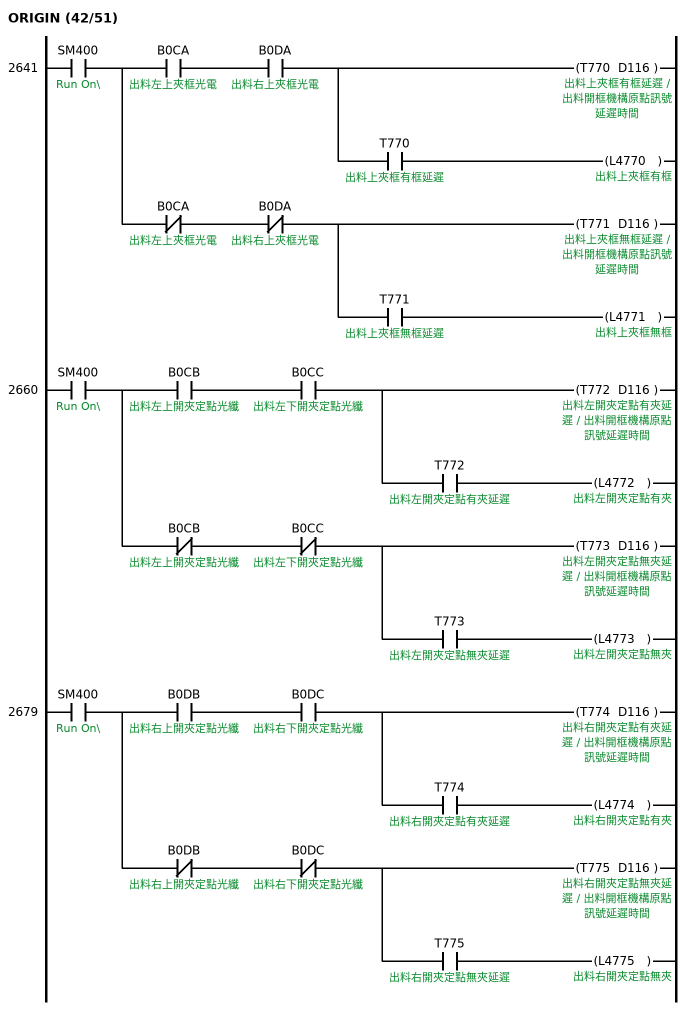
[picture p456: ladder of ORIGIN, rungs at steps 2641 to 2679]
2641  LD      SM400  ; Run On\
      MPS
      AND     B0CA  ; 出料左上夾框光電
      AND     B0DA  ; 出料右上夾框光電
      OUT     T770 D116  ; 出料上夾框有框延遲 / 出料開框機構原點訊號延遲時間
      AND     T770  ; 出料上夾框有框延遲
      OUT     L4770  ; 出料上夾框有框
      MPP
      ANI     B0CA  ; 出料左上夾框光電
      ANI     B0DA  ; 出料右上夾框光電
      OUT     T771 D116  ; 出料上夾框無框延遲 / 出料開框機構原點訊號延遲時間
      AND     T771  ; 出料上夾框無框延遲
      OUT     L4771  ; 出料上夾框無框
2660  LD      SM400  ; Run On\
      MPS
      AND     B0CB  ; 出料左上開夾定點光纖
      AND     B0CC  ; 出料左下開夾定點光纖
      OUT     T772 D116  ; 出料左開夾定點有夾延遲 / 出料開框機構原點訊號延遲時間
      AND     T772  ; 出料左開夾定點有夾延遲
      OUT     L4772  ; 出料左開夾定點有夾
      MPP
      ANI     B0CB  ; 出料左上開夾定點光纖
      ANI     B0CC  ; 出料左下開夾定點光纖
      OUT     T773 D116  ; 出料左開夾定點無夾延遲 / 出料開框機構原點訊號延遲時間
      AND     T773  ; 出料左開夾定點無夾延遲
      OUT     L4773  ; 出料左開夾定點無夾
2679  LD      SM400  ; Run On\
      MPS
      AND     B0DB  ; 出料右上開夾定點光纖
      AND     B0DC  ; 出料右下開夾定點光纖
      OUT     T774 D116  ; 出料右開夾定點有夾延遲 / 出料開框機構原點訊號延遲時間
      AND     T774  ; 出料右開夾定點有夾延遲
      OUT     L4774  ; 出料右開夾定點有夾
      MPP
      ANI     B0DB  ; 出料右上開夾定點光纖
      ANI     B0DC  ; 出料右下開夾定點光纖
      OUT     T775 D116  ; 出料右開夾定點無夾延遲 / 出料開框機構原點訊號延遲時間
      AND     T775  ; 出料右開夾定點無夾延遲
      OUT     L4775  ; 出料右開夾定點無夾
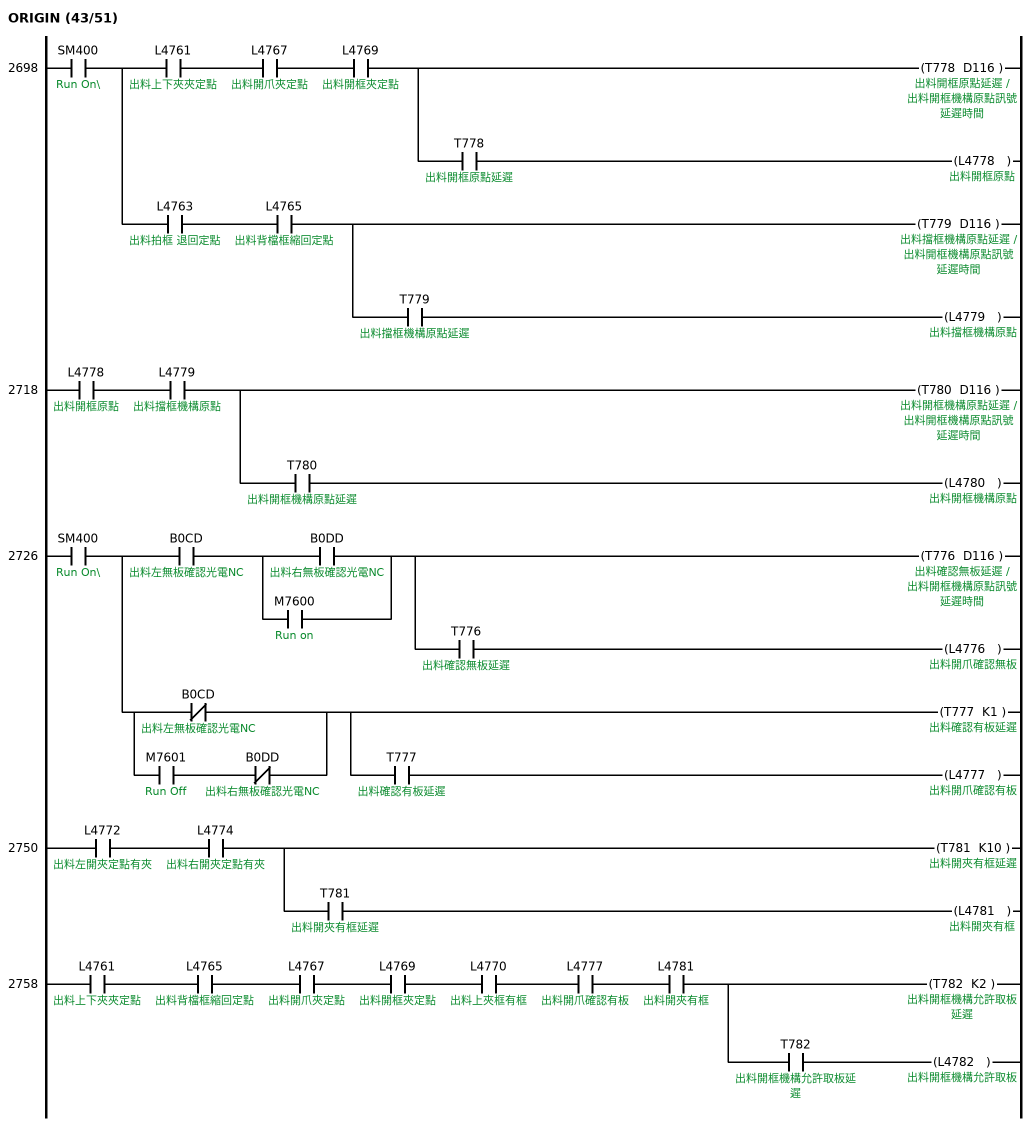
2698  LD      SM400  ; Run On\
      MPS
      AND     L4761  ; 出料上下夾夾定點
      AND     L4767  ; 出料開爪夾定點
      AND     L4769  ; 出料開框夾定點
      OUT     T778 D116  ; 出料開框原點延遲 / 出料開框機構原點訊號延遲時間
      AND     T778  ; 出料開框原點延遲
      OUT     L4778  ; 出料開框原點
      MPP
      AND     L4763  ; 出料拍框 退回定點
      AND     L4765  ; 出料背檔框縮回定點
      OUT     T779 D116  ; 出料擋框機構原點延遲 / 出料開框機構原點訊號延遲時間
      AND     T779  ; 出料擋框機構原點延遲
      OUT     L4779  ; 出料擋框機構原點
2718  LD      L4778  ; 出料開框原點
      AND     L4779  ; 出料擋框機構原點
      OUT     T780 D116  ; 出料開框機構原點延遲 / 出料開框機構原點訊號延遲時間
      AND     T780  ; 出料開框機構原點延遲
      OUT     L4780  ; 出料開框機構原點
2726  LD      SM400  ; Run On\
      MPS
      AND     B0CD  ; 出料左無板確認光電NC
      LD      B0DD  ; 出料右無板確認光電NC
      OR      M7600  ; Run on
      ANB
      OUT     T776 D116  ; 出料確認無板延遲 / 出料開框機構原點訊號延遲時間
      AND     T776  ; 出料確認無板延遲
      OUT     L4776  ; 出料開爪確認無板
      MPP
      LDI     B0CD  ; 出料左無板確認光電NC
      LD      M7601  ; Run Off
      ANI     B0DD  ; 出料右無板確認光電NC
      ORB
      ANB
      OUT     T777 K1  ; 出料確認有板延遲
      AND     T777  ; 出料確認有板延遲
      OUT     L4777  ; 出料開爪確認有板
2750  LD      L4772  ; 出料左開夾定點有夾
      AND     L4774  ; 出料右開夾定點有夾
      OUT     T781 K10  ; 出料開夾有框延遲
      AND     T781  ; 出料開夾有框延遲
      OUT     L4781  ; 出料開夾有框
2758  LD      L4761  ; 出料上下夾夾定點
      AND     L4765  ; 出料背檔框縮回定點
      AND     L4767  ; 出料開爪夾定點
      AND     L4769  ; 出料開框夾定點
      AND     L4770  ; 出料上夾框有框
      AND     L4777  ; 出料開爪確認有板
      AND     L4781  ; 出料開夾有框
      OUT     T782 K2  ; 出料開框機構允許取板延遲
      AND     T782  ; 出料開框機構允許取板延遲
      OUT     L4782  ; 出料開框機構允許取板
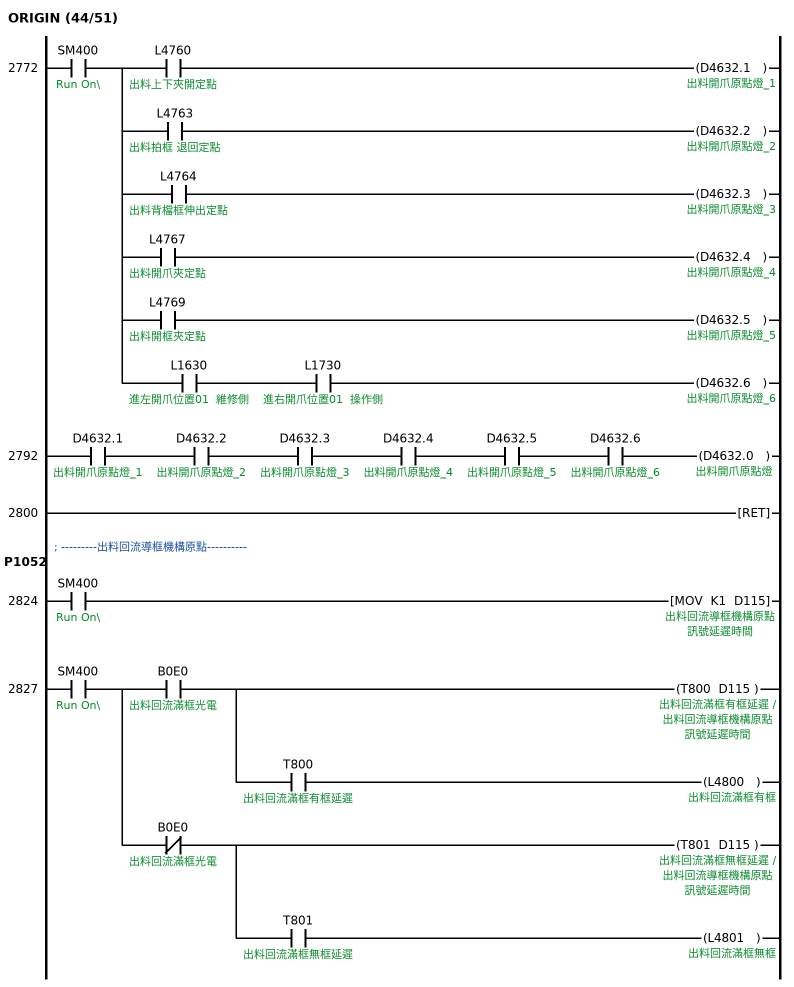
2772  LD      SM400  ; Run On\
      MPS
      AND     L4760  ; 出料上下夾開定點
      OUT     D4632.1  ; 出料開爪原點燈_1
      MRD
      AND     L4763  ; 出料拍框 退回定點
      OUT     D4632.2  ; 出料開爪原點燈_2
      MRD
      AND     L4764  ; 出料背檔框伸出定點
      OUT     D4632.3  ; 出料開爪原點燈_3
      MRD
      AND     L4767  ; 出料開爪夾定點
      OUT     D4632.4  ; 出料開爪原點燈_4
      MRD
      AND     L4769  ; 出料開框夾定點
      OUT     D4632.5  ; 出料開爪原點燈_5
      MPP
      AND     L1630  ; 進左開爪位置01  維修側
      AND     L1730  ; 進右開爪位置01  操作側
      OUT     D4632.6  ; 出料開爪原點燈_6
2792  LD      D4632.1  ; 出料開爪原點燈_1
      AND     D4632.2  ; 出料開爪原點燈_2
      AND     D4632.3  ; 出料開爪原點燈_3
      AND     D4632.4  ; 出料開爪原點燈_4
      AND     D4632.5  ; 出料開爪原點燈_5
      AND     D4632.6  ; 出料開爪原點燈_6
      OUT     D4632.0  ; 出料開爪原點燈
2800  RET
; ---------出料回流導框機構原點----------
      P1052
2824  LD      SM400  ; Run On\
      MOV     K1 D115  ; 出料回流導框機構原點訊號延遲時間
2827  LD      SM400  ; Run On\
      MPS
      AND     B0E0  ; 出料回流滿框光電
      OUT     T800 D115  ; 出料回流滿框有框延遲 / 出料回流導框機構原點訊號延遲時間
      AND     T800  ; 出料回流滿框有框延遲
      OUT     L4800  ; 出料回流滿框有框
      MPP
      ANI     B0E0  ; 出料回流滿框光電
      OUT     T801 D115  ; 出料回流滿框無框延遲 / 出料回流導框機構原點訊號延遲時間
      AND     T801  ; 出料回流滿框無框延遲
      OUT     L4801  ; 出料回流滿框無框
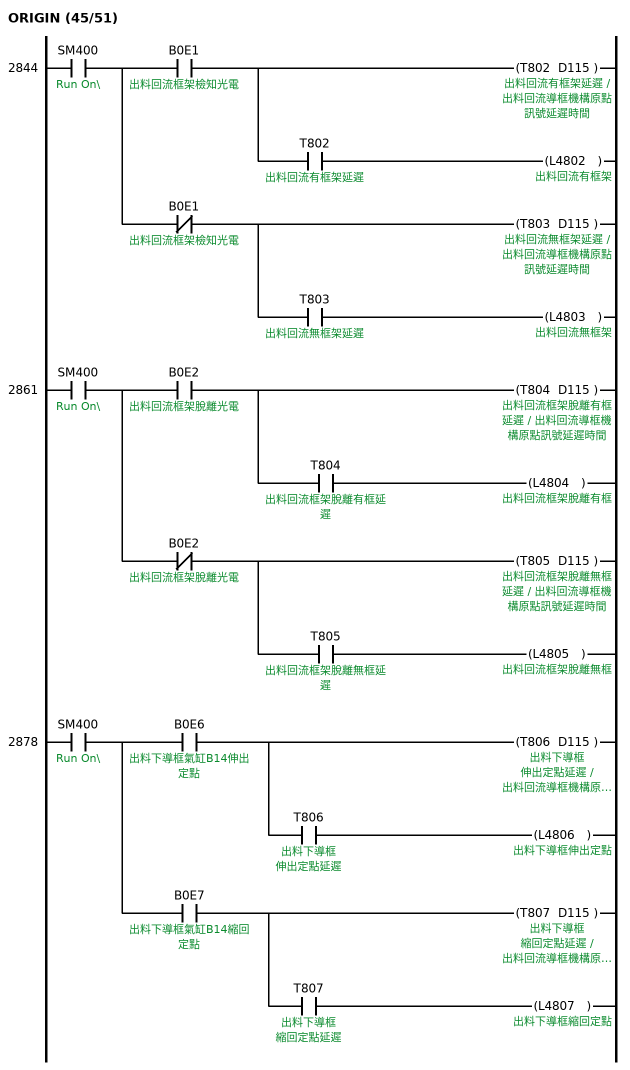
2844  LD      SM400  ; Run On\
      MPS
      AND     B0E1  ; 出料回流框架檢知光電
      OUT     T802 D115  ; 出料回流有框架延遲 / 出料回流導框機構原點訊號延遲時間
      AND     T802  ; 出料回流有框架延遲
      OUT     L4802  ; 出料回流有框架
      MPP
      ANI     B0E1  ; 出料回流框架檢知光電
      OUT     T803 D115  ; 出料回流無框架延遲 / 出料回流導框機構原點訊號延遲時間
      AND     T803  ; 出料回流無框架延遲
      OUT     L4803  ; 出料回流無框架
2861  LD      SM400  ; Run On\
      MPS
      AND     B0E2  ; 出料回流框架脫離光電
      OUT     T804 D115  ; 出料回流框架脫離有框延遲 / 出料回流導框機構原點訊號延遲時間
      AND     T804  ; 出料回流框架脫離有框延遲
      OUT     L4804  ; 出料回流框架脫離有框
      MPP
      ANI     B0E2  ; 出料回流框架脫離光電
      OUT     T805 D115  ; 出料回流框架脫離無框延遲 / 出料回流導框機構原點訊號延遲時間
      AND     T805  ; 出料回流框架脫離無框延遲
      OUT     L4805  ; 出料回流框架脫離無框
2878  LD      SM400  ; Run On\
      MPS
      AND     B0E6  ; 出料下導框氣缸B14伸出定點
      OUT     T806 D115  ; 出料下導框    伸出定點延遲 / 出料回流導框機構原點訊號延遲時間
      AND     T806  ; 出料下導框    伸出定點延遲
      OUT     L4806  ; 出料下導框伸出定點
      MPP
      AND     B0E7  ; 出料下導框氣缸B14縮回定點
      OUT     T807 D115  ; 出料下導框    縮回定點延遲 / 出料回流導框機構原點訊號延遲時間
      AND     T807  ; 出料下導框    縮回定點延遲
      OUT     L4807  ; 出料下導框縮回定點
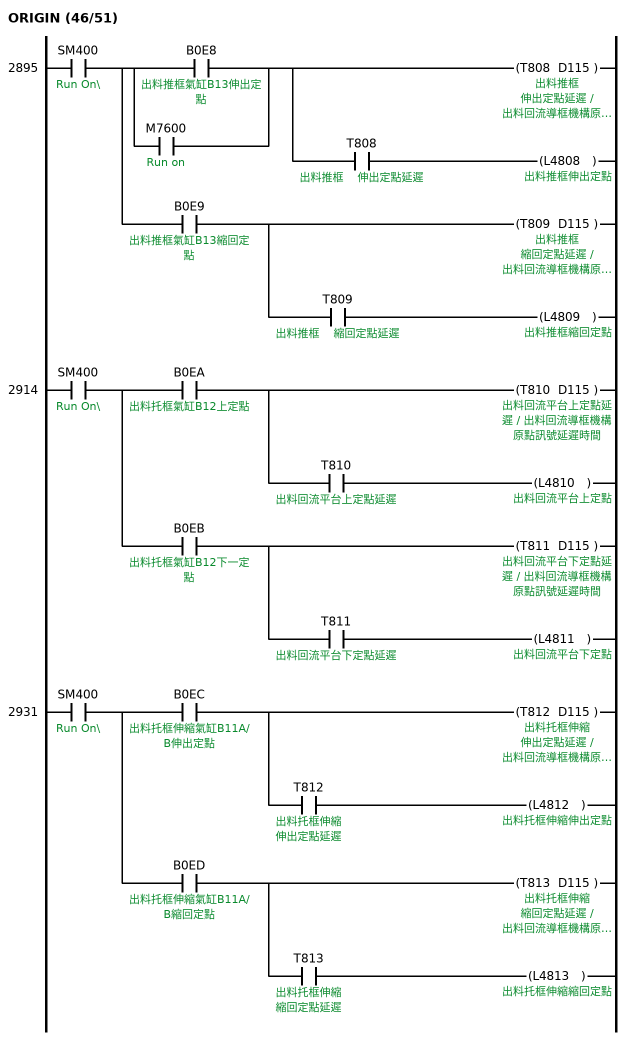
2895  LD      SM400  ; Run On\
      MPS
      LD      B0E8  ; 出料推框氣缸B13伸出定點
      OR      M7600  ; Run on
      ANB
      OUT     T808 D115  ; 出料推框    伸出定點延遲 / 出料回流導框機構原點訊號延遲時間
      AND     T808  ; 出料推框    伸出定點延遲
      OUT     L4808  ; 出料推框伸出定點
      MPP
      AND     B0E9  ; 出料推框氣缸B13縮回定點
      OUT     T809 D115  ; 出料推框    縮回定點延遲 / 出料回流導框機構原點訊號延遲時間
      AND     T809  ; 出料推框    縮回定點延遲
      OUT     L4809  ; 出料推框縮回定點
2914  LD      SM400  ; Run On\
      MPS
      AND     B0EA  ; 出料托框氣缸B12上定點
      OUT     T810 D115  ; 出料回流平台上定點延遲 / 出料回流導框機構原點訊號延遲時間
      AND     T810  ; 出料回流平台上定點延遲
      OUT     L4810  ; 出料回流平台上定點
      MPP
      AND     B0EB  ; 出料托框氣缸B12下一定點
      OUT     T811 D115  ; 出料回流平台下定點延遲 / 出料回流導框機構原點訊號延遲時間
      AND     T811  ; 出料回流平台下定點延遲
      OUT     L4811  ; 出料回流平台下定點
2931  LD      SM400  ; Run On\
      MPS
      AND     B0EC  ; 出料托框伸縮氣缸B11A/B伸出定點
      OUT     T812 D115  ; 出料托框伸縮    伸出定點延遲 / 出料回流導框機構原點訊號延遲時間
      AND     T812  ; 出料托框伸縮    伸出定點延遲
      OUT     L4812  ; 出料托框伸縮伸出定點
      MPP
      AND     B0ED  ; 出料托框伸縮氣缸B11A/B縮回定點
      OUT     T813 D115  ; 出料托框伸縮    縮回定點延遲 / 出料回流導框機構原點訊號延遲時間
      AND     T813  ; 出料托框伸縮    縮回定點延遲
      OUT     L4813  ; 出料托框伸縮縮回定點
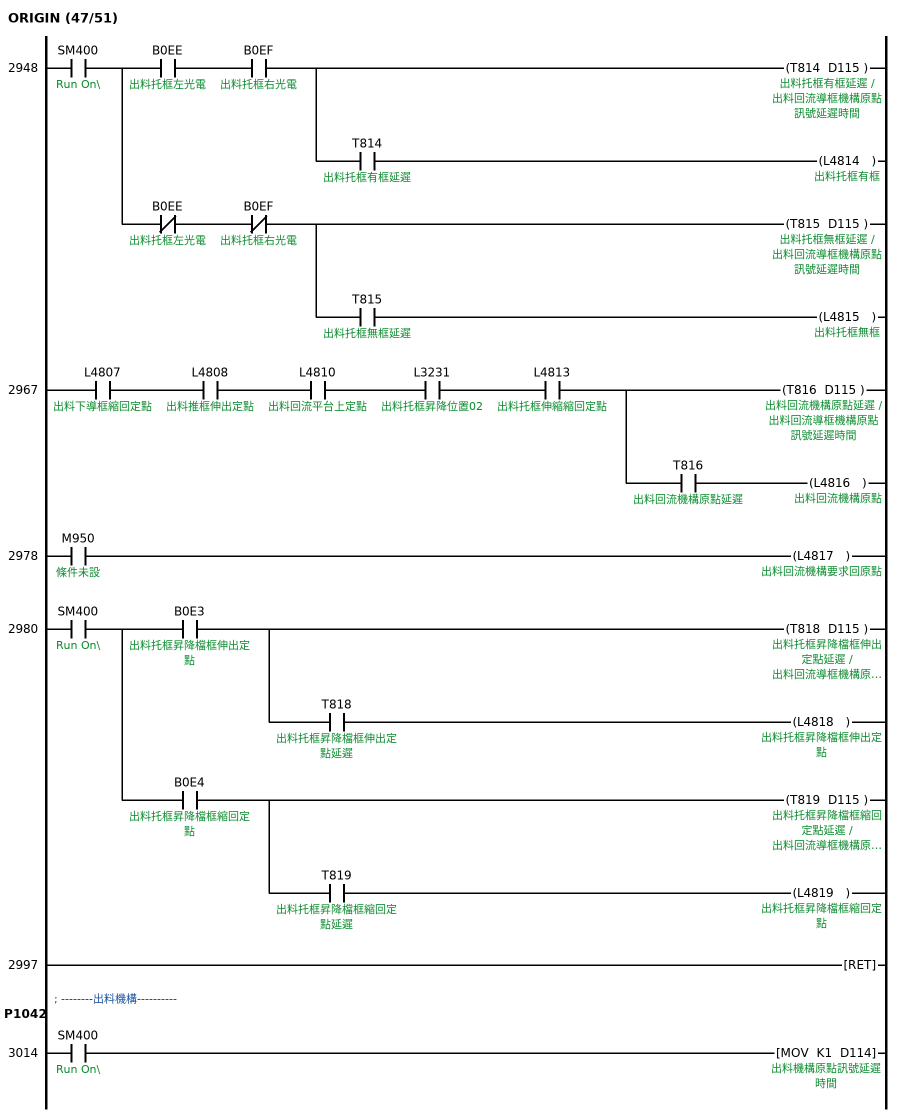
2948  LD      SM400  ; Run On\
      MPS
      AND     B0EE  ; 出料托框左光電
      AND     B0EF  ; 出料托框右光電
      OUT     T814 D115  ; 出料托框有框延遲 / 出料回流導框機構原點訊號延遲時間
      AND     T814  ; 出料托框有框延遲
      OUT     L4814  ; 出料托框有框
      MPP
      ANI     B0EE  ; 出料托框左光電
      ANI     B0EF  ; 出料托框右光電
      OUT     T815 D115  ; 出料托框無框延遲 / 出料回流導框機構原點訊號延遲時間
      AND     T815  ; 出料托框無框延遲
      OUT     L4815  ; 出料托框無框
2967  LD      L4807  ; 出料下導框縮回定點
      AND     L4808  ; 出料推框伸出定點
      AND     L4810  ; 出料回流平台上定點
      AND     L3231  ; 出料托框昇降位置02
      AND     L4813  ; 出料托框伸縮縮回定點
      OUT     T816 D115  ; 出料回流機構原點延遲 / 出料回流導框機構原點訊號延遲時間
      AND     T816  ; 出料回流機構原點延遲
      OUT     L4816  ; 出料回流機構原點
2978  LD      M950  ; 條件未設
      OUT     L4817  ; 出料回流機構要求回原點
2980  LD      SM400  ; Run On\
      MPS
      AND     B0E3  ; 出料托框昇降檔框伸出定點
      OUT     T818 D115  ; 出料托框昇降檔框伸出定點延遲 / 出料回流導框機構原點訊號延遲時間
      AND     T818  ; 出料托框昇降檔框伸出定點延遲
      OUT     L4818  ; 出料托框昇降檔框伸出定點
      MPP
      AND     B0E4  ; 出料托框昇降檔框縮回定點
      OUT     T819 D115  ; 出料托框昇降檔框縮回定點延遲 / 出料回流導框機構原點訊號延遲時間
      AND     T819  ; 出料托框昇降檔框縮回定點延遲
      OUT     L4819  ; 出料托框昇降檔框縮回定點
2997  RET
; --------出料機構----------
      P1042
3014  LD      SM400  ; Run On\
      MOV     K1 D114  ; 出料機構原點訊號延遲時間
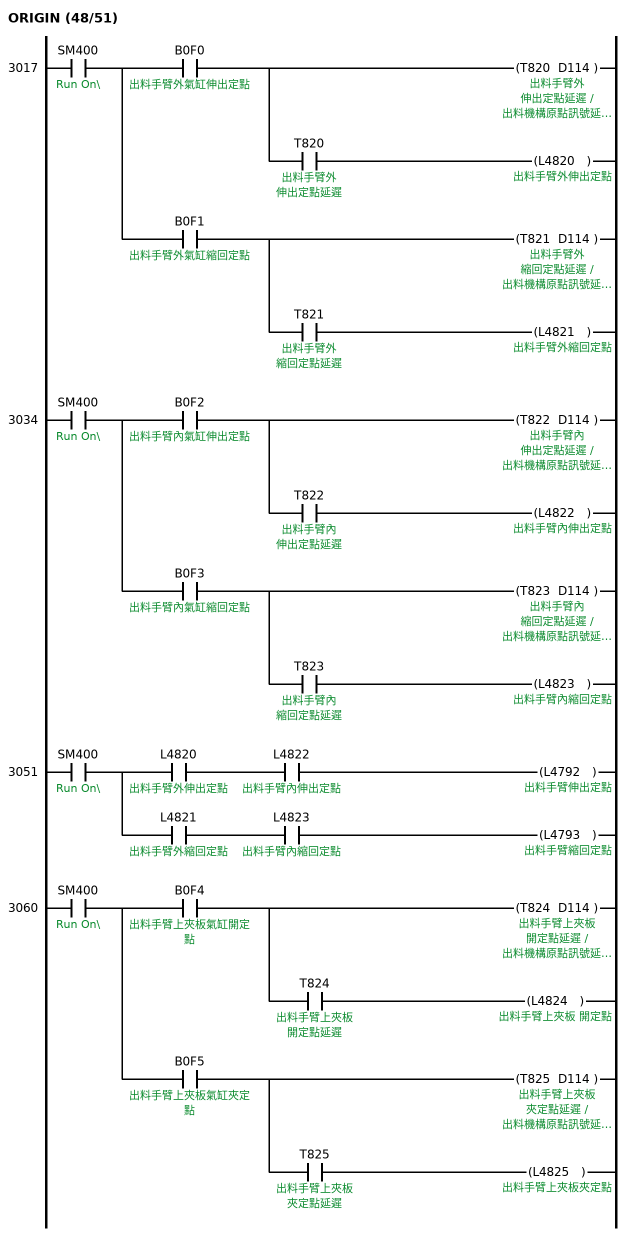
3017  LD      SM400  ; Run On\
      MPS
      AND     B0F0  ; 出料手臂外氣缸伸出定點
      OUT     T820 D114  ; 出料手臂外    伸出定點延遲 / 出料機構原點訊號延遲時間
      AND     T820  ; 出料手臂外    伸出定點延遲
      OUT     L4820  ; 出料手臂外伸出定點
      MPP
      AND     B0F1  ; 出料手臂外氣缸縮回定點
      OUT     T821 D114  ; 出料手臂外    縮回定點延遲 / 出料機構原點訊號延遲時間
      AND     T821  ; 出料手臂外    縮回定點延遲
      OUT     L4821  ; 出料手臂外縮回定點
3034  LD      SM400  ; Run On\
      MPS
      AND     B0F2  ; 出料手臂內氣缸伸出定點
      OUT     T822 D114  ; 出料手臂內    伸出定點延遲 / 出料機構原點訊號延遲時間
      AND     T822  ; 出料手臂內    伸出定點延遲
      OUT     L4822  ; 出料手臂內伸出定點
      MPP
      AND     B0F3  ; 出料手臂內氣缸縮回定點
      OUT     T823 D114  ; 出料手臂內    縮回定點延遲 / 出料機構原點訊號延遲時間
      AND     T823  ; 出料手臂內    縮回定點延遲
      OUT     L4823  ; 出料手臂內縮回定點
3051  LD      SM400  ; Run On\
      MPS
      AND     L4820  ; 出料手臂外伸出定點
      AND     L4822  ; 出料手臂內伸出定點
      OUT     L4792  ; 出料手臂伸出定點
      MPP
      AND     L4821  ; 出料手臂外縮回定點
      AND     L4823  ; 出料手臂內縮回定點
      OUT     L4793  ; 出料手臂縮回定點
3060  LD      SM400  ; Run On\
      MPS
      AND     B0F4  ; 出料手臂上夾板氣缸開定點
      OUT     T824 D114  ; 出料手臂上夾板    開定點延遲 / 出料機構原點訊號延遲時間
      AND     T824  ; 出料手臂上夾板    開定點延遲
      OUT     L4824  ; 出料手臂上夾板 開定點
      MPP
      AND     B0F5  ; 出料手臂上夾板氣缸夾定點
      OUT     T825 D114  ; 出料手臂上夾板    夾定點延遲 / 出料機構原點訊號延遲時間
      AND     T825  ; 出料手臂上夾板    夾定點延遲
      OUT     L4825  ; 出料手臂上夾板夾定點
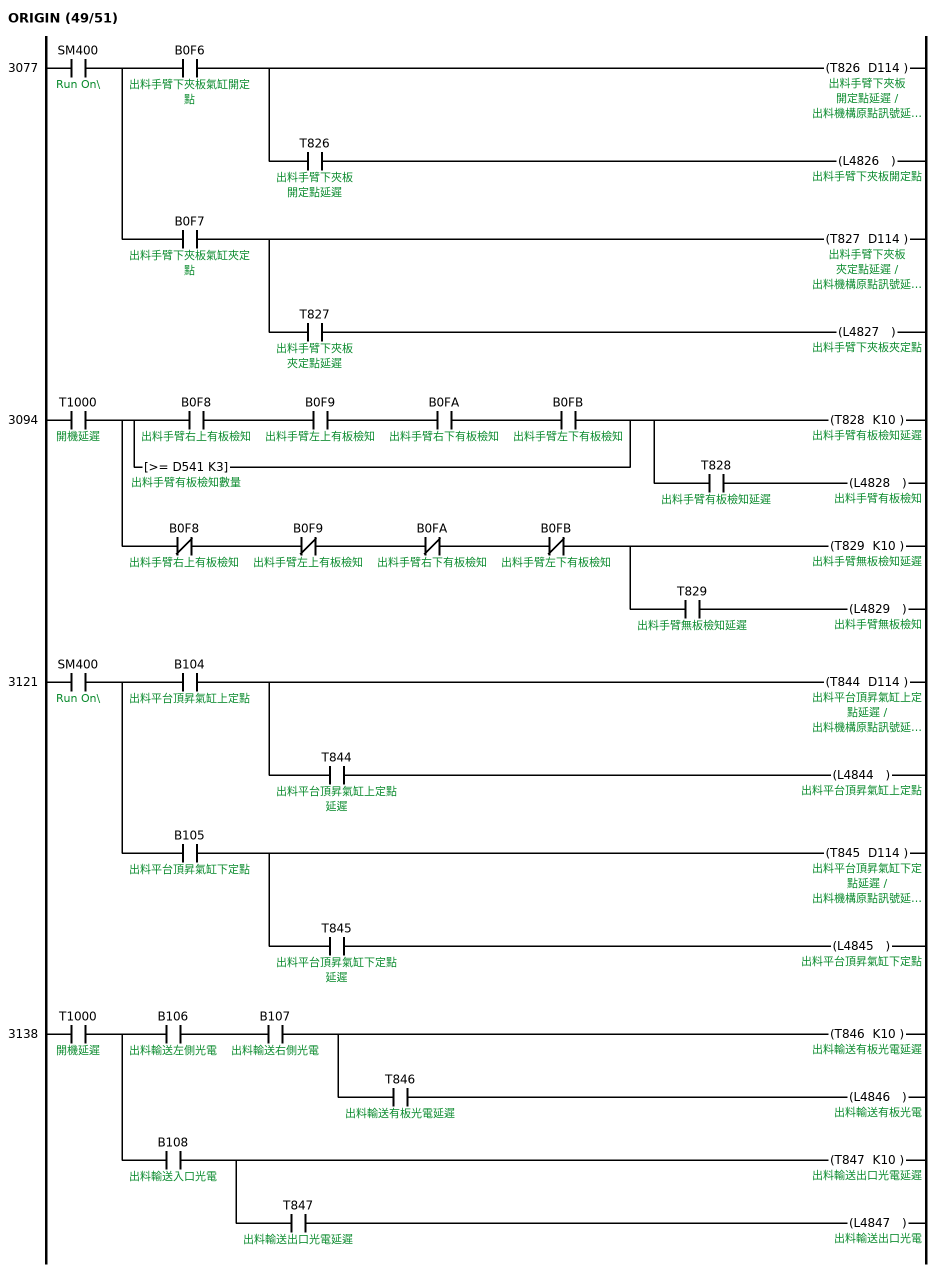
3077  LD      SM400  ; Run On\
      MPS
      AND     B0F6  ; 出料手臂下夾板氣缸開定點
      OUT     T826 D114  ; 出料手臂下夾板    開定點延遲 / 出料機構原點訊號延遲時間
      AND     T826  ; 出料手臂下夾板    開定點延遲
      OUT     L4826  ; 出料手臂下夾板開定點
      MPP
      AND     B0F7  ; 出料手臂下夾板氣缸夾定點
      OUT     T827 D114  ; 出料手臂下夾板    夾定點延遲 / 出料機構原點訊號延遲時間
      AND     T827  ; 出料手臂下夾板    夾定點延遲
      OUT     L4827  ; 出料手臂下夾板夾定點
3094  LD      T1000  ; 開機延遲
      MPS
      LD      B0F8  ; 出料手臂右上有板檢知
      AND     B0F9  ; 出料手臂左上有板檢知
      AND     B0FA  ; 出料手臂右下有板檢知
      AND     B0FB  ; 出料手臂左下有板檢知
      OR>=    D541 K3  ; 出料手臂有板檢知數量
      ANB
      OUT     T828 K10  ; 出料手臂有板檢知延遲
      AND     T828  ; 出料手臂有板檢知延遲
      OUT     L4828  ; 出料手臂有板檢知
      MPP
      ANI     B0F8  ; 出料手臂右上有板檢知
      ANI     B0F9  ; 出料手臂左上有板檢知
      ANI     B0FA  ; 出料手臂右下有板檢知
      ANI     B0FB  ; 出料手臂左下有板檢知
      OUT     T829 K10  ; 出料手臂無板檢知延遲
      AND     T829  ; 出料手臂無板檢知延遲
      OUT     L4829  ; 出料手臂無板檢知
3121  LD      SM400  ; Run On\
      MPS
      AND     B104  ; 出料平台頂昇氣缸上定點
      OUT     T844 D114  ; 出料平台頂昇氣缸上定點延遲 / 出料機構原點訊號延遲時間
      AND     T844  ; 出料平台頂昇氣缸上定點延遲
      OUT     L4844  ; 出料平台頂昇氣缸上定點
      MPP
      AND     B105  ; 出料平台頂昇氣缸下定點
      OUT     T845 D114  ; 出料平台頂昇氣缸下定點延遲 / 出料機構原點訊號延遲時間
      AND     T845  ; 出料平台頂昇氣缸下定點延遲
      OUT     L4845  ; 出料平台頂昇氣缸下定點
3138  LD      T1000  ; 開機延遲
      MPS
      AND     B106  ; 出料輸送左側光電
      AND     B107  ; 出料輸送右側光電
      OUT     T846 K10  ; 出料輸送有板光電延遲
      AND     T846  ; 出料輸送有板光電延遲
      OUT     L4846  ; 出料輸送有板光電
      MPP
      AND     B108  ; 出料輸送入口光電
      OUT     T847 K10  ; 出料輸送出口光電延遲
      AND     T847  ; 出料輸送出口光電延遲
      OUT     L4847  ; 出料輸送出口光電
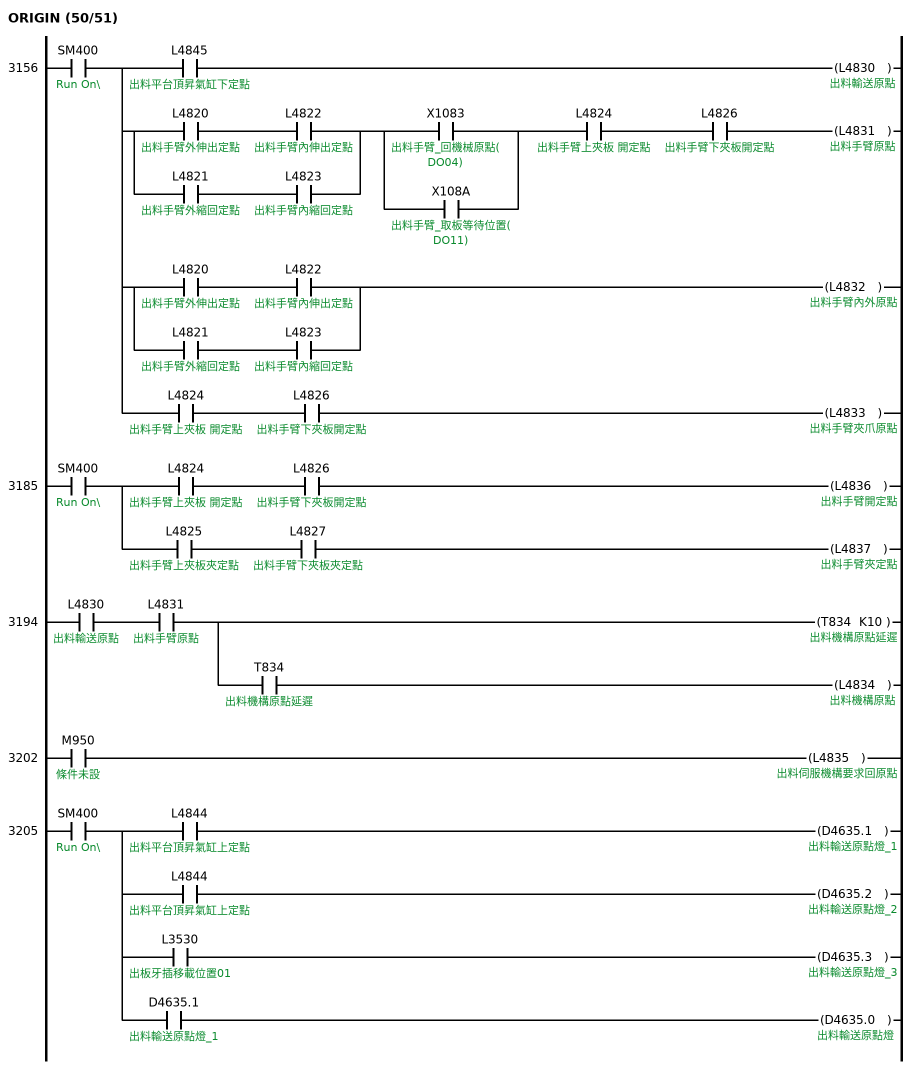
3156  LD      SM400  ; Run On\
      MPS
      AND     L4845  ; 出料平台頂昇氣缸下定點
      OUT     L4830  ; 出料輸送原點
      MRD
      LD      L4820  ; 出料手臂外伸出定點
      AND     L4822  ; 出料手臂內伸出定點
      LD      L4821  ; 出料手臂外縮回定點
      AND     L4823  ; 出料手臂內縮回定點
      ORB
      ANB
      LD      X1083  ; 出料手臂_回機械原點(DO04)
      OR      X108A  ; 出料手臂_取板等待位置(DO11)
      ANB
      AND     L4824  ; 出料手臂上夾板 開定點
      AND     L4826  ; 出料手臂下夾板開定點
      OUT     L4831  ; 出料手臂原點
      MRD
      LD      L4820  ; 出料手臂外伸出定點
      AND     L4822  ; 出料手臂內伸出定點
      LD      L4821  ; 出料手臂外縮回定點
      AND     L4823  ; 出料手臂內縮回定點
      ORB
      ANB
      OUT     L4832  ; 出料手臂內外原點
      MPP
      AND     L4824  ; 出料手臂上夾板 開定點
      AND     L4826  ; 出料手臂下夾板開定點
      OUT     L4833  ; 出料手臂夾爪原點
3185  LD      SM400  ; Run On\
      MPS
      AND     L4824  ; 出料手臂上夾板 開定點
      AND     L4826  ; 出料手臂下夾板開定點
      OUT     L4836  ; 出料手臂開定點
      MPP
      AND     L4825  ; 出料手臂上夾板夾定點
      AND     L4827  ; 出料手臂下夾板夾定點
      OUT     L4837  ; 出料手臂夾定點
3194  LD      L4830  ; 出料輸送原點
      AND     L4831  ; 出料手臂原點
      OUT     T834 K10  ; 出料機構原點延遲
      AND     T834  ; 出料機構原點延遲
      OUT     L4834  ; 出料機構原點
3202  LD      M950  ; 條件未設
      OUT     L4835  ; 出料伺服機構要求回原點
3205  LD      SM400  ; Run On\
      MPS
      AND     L4844  ; 出料平台頂昇氣缸上定點
      OUT     D4635.1  ; 出料輸送原點燈_1
      MRD
      AND     L4844  ; 出料平台頂昇氣缸上定點
      OUT     D4635.2  ; 出料輸送原點燈_2
      MRD
      AND     L3530  ; 出板牙插移載位置01
      OUT     D4635.3  ; 出料輸送原點燈_3
      MPP
      AND     D4635.1  ; 出料輸送原點燈_1
      OUT     D4635.0  ; 出料輸送原點燈
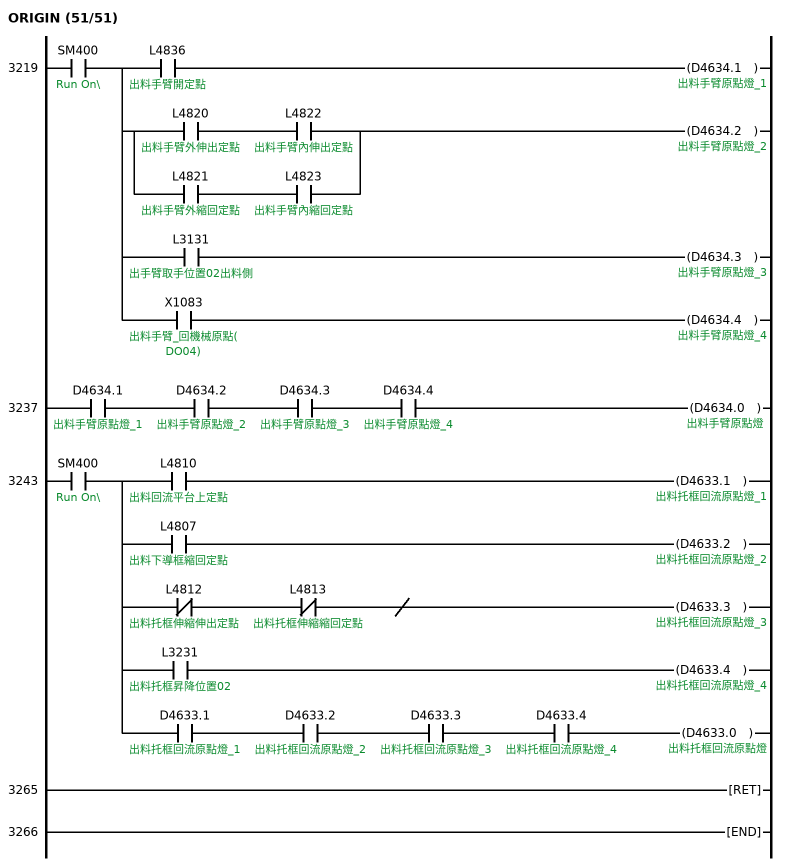
3219  LD      SM400  ; Run On\
      MPS
      AND     L4836  ; 出料手臂開定點
      OUT     D4634.1  ; 出料手臂原點燈_1
      MRD
      LD      L4820  ; 出料手臂外伸出定點
      AND     L4822  ; 出料手臂內伸出定點
      LD      L4821  ; 出料手臂外縮回定點
      AND     L4823  ; 出料手臂內縮回定點
      ORB
      ANB
      OUT     D4634.2  ; 出料手臂原點燈_2
      MRD
      AND     L3131  ; 出手臂取手位置02出料側
      OUT     D4634.3  ; 出料手臂原點燈_3
      MPP
      AND     X1083  ; 出料手臂_回機械原點(DO04)
      OUT     D4634.4  ; 出料手臂原點燈_4
3237  LD      D4634.1  ; 出料手臂原點燈_1
      AND     D4634.2  ; 出料手臂原點燈_2
      AND     D4634.3  ; 出料手臂原點燈_3
      AND     D4634.4  ; 出料手臂原點燈_4
      OUT     D4634.0  ; 出料手臂原點燈
3243  LD      SM400  ; Run On\
      MPS
      AND     L4810  ; 出料回流平台上定點
      OUT     D4633.1  ; 出料托框回流原點燈_1
      MRD
      AND     L4807  ; 出料下導框縮回定點
      OUT     D4633.2  ; 出料托框回流原點燈_2
      MRD
      ANI     L4812  ; 出料托框伸縮伸出定點
      ANI     L4813  ; 出料托框伸縮縮回定點
      INV
      OUT     D4633.3  ; 出料托框回流原點燈_3
      MRD
      AND     L3231  ; 出料托框昇降位置02
      OUT     D4633.4  ; 出料托框回流原點燈_4
      MPP
      AND     D4633.1  ; 出料托框回流原點燈_1
      AND     D4633.2  ; 出料托框回流原點燈_2
      AND     D4633.3  ; 出料托框回流原點燈_3
      AND     D4633.4  ; 出料托框回流原點燈_4
      OUT     D4633.0  ; 出料托框回流原點燈
3265  RET
3266  END
END_PROGRAM

PROGRAM SECS
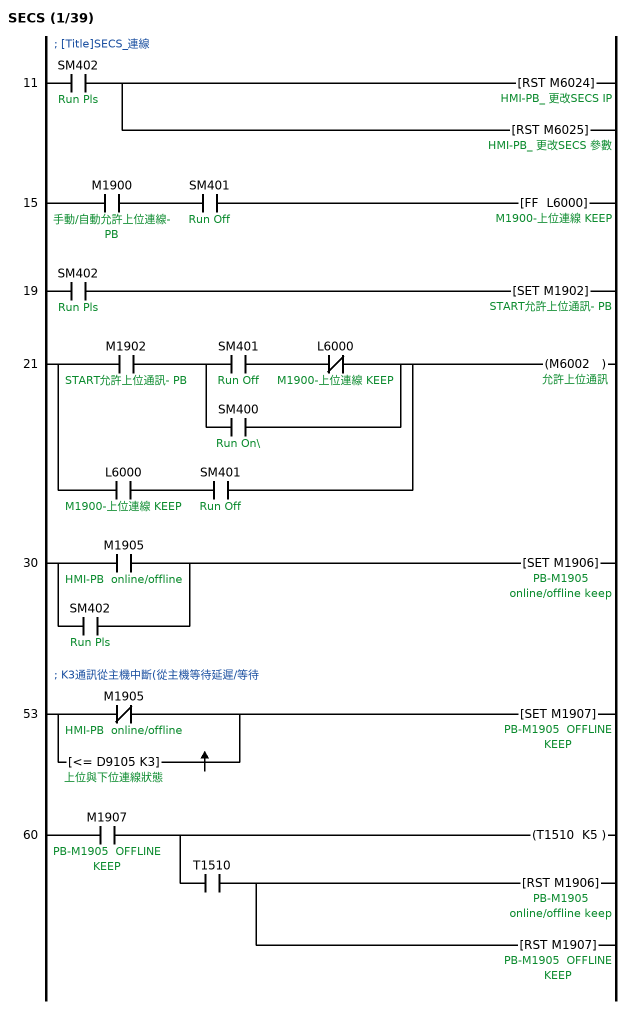
; [Title]SECS_連線
11    LD      SM402  ; Run Pls
      RST     M6024  ; HMI-PB_ 更改SECS IP
      RST     M6025  ; HMI-PB_ 更改SECS 參數
15    LD      M1900  ; 手動/自動允許上位連線-PB
      AND     SM401  ; Run Off
      FF      L6000  ; M1900-上位連線 KEEP
19    LD      SM402  ; Run Pls
      SET     M1902  ; START允許上位通訊- PB
21    LD      M1902  ; START允許上位通訊- PB
      LD      SM401  ; Run Off
      ANI     L6000  ; M1900-上位連線 KEEP
      OR      SM400  ; Run On\
      ANB
      LD      L6000  ; M1900-上位連線 KEEP
      AND     SM401  ; Run Off
      ORB
      OUT     M6002  ; 允許上位通訊
30    LD      M1905  ; HMI-PB  online/offline
      OR      SM402  ; Run Pls
      SET     M1906  ; PB-M1905  online/offline keep
; K3通訊從主機中斷(從主機等待延遲/等待
53    LDI     M1905  ; HMI-PB  online/offline
      LD<=    D9105 K3  ; 上位與下位連線狀態
      MEP
      ORB
      SET     M1907  ; PB-M1905  OFFLINE KEEP
60    LD      M1907  ; PB-M1905  OFFLINE KEEP
      OUT     T1510 K5
      AND     T1510
      RST     M1906  ; PB-M1905  online/offline keep
      RST     M1907  ; PB-M1905  OFFLINE KEEP
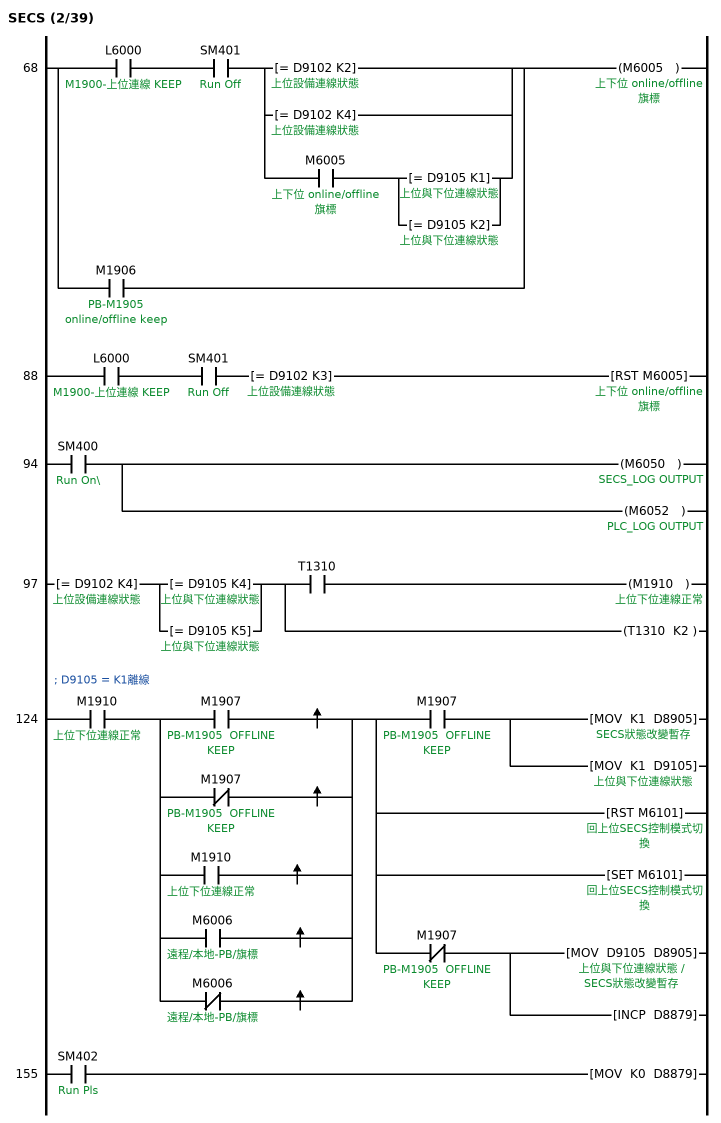
68    LD      L6000  ; M1900-上位連線 KEEP
      AND     SM401  ; Run Off
      LD=     D9102 K2  ; 上位設備連線狀態
      OR=     D9102 K4  ; 上位設備連線狀態
      LD      M6005  ; 上下位 online/offline 旗標
      LD=     D9105 K1  ; 上位與下位連線狀態
      OR=     D9105 K2  ; 上位與下位連線狀態
      ANB
      ORB
      ANB
      OR      M1906  ; PB-M1905  online/offline keep
      OUT     M6005  ; 上下位 online/offline 旗標
88    LD      L6000  ; M1900-上位連線 KEEP
      AND     SM401  ; Run Off
      AND=    D9102 K3  ; 上位設備連線狀態
      RST     M6005  ; 上下位 online/offline 旗標
94    LD      SM400  ; Run On\
      OUT     M6050  ; SECS_LOG OUTPUT
      OUT     M6052  ; PLC_LOG OUTPUT
97    LD=     D9102 K4  ; 上位設備連線狀態
      LD=     D9105 K4  ; 上位與下位連線狀態
      OR=     D9105 K5  ; 上位與下位連線狀態
      ANB
      MPS
      AND     T1310
      OUT     M1910  ; 上位下位連線正常
      MPP
      OUT     T1310 K2
; D9105 = K1離線
124   LD      M1910  ; 上位下位連線正常
      LD      M1907  ; PB-M1905  OFFLINE KEEP
      MEP
      LDI     M1907  ; PB-M1905  OFFLINE KEEP
      MEP
      ORB
      LD      M1910  ; 上位下位連線正常
      MEP
      ORB
      LD      M6006  ; 遠程/本地-PB/旗標
      MEP
      ORB
      LDI     M6006  ; 遠程/本地-PB/旗標
      MEP
      ORB
      ANB
      MPS
      AND     M1907  ; PB-M1905  OFFLINE KEEP
      MOV     K1 D8905  ; SECS狀態改變暫存
      MOV     K1 D9105
      MPP
      RST     M6101  ; 回上位SECS控制模式切換
      SET     M6101  ; 回上位SECS控制模式切換
      ANI     M1907  ; PB-M1905  OFFLINE KEEP
      MOV     D9105 D8905
      INCP    D8879
155   LD      SM402  ; Run Pls
      MOV     K0 D8879
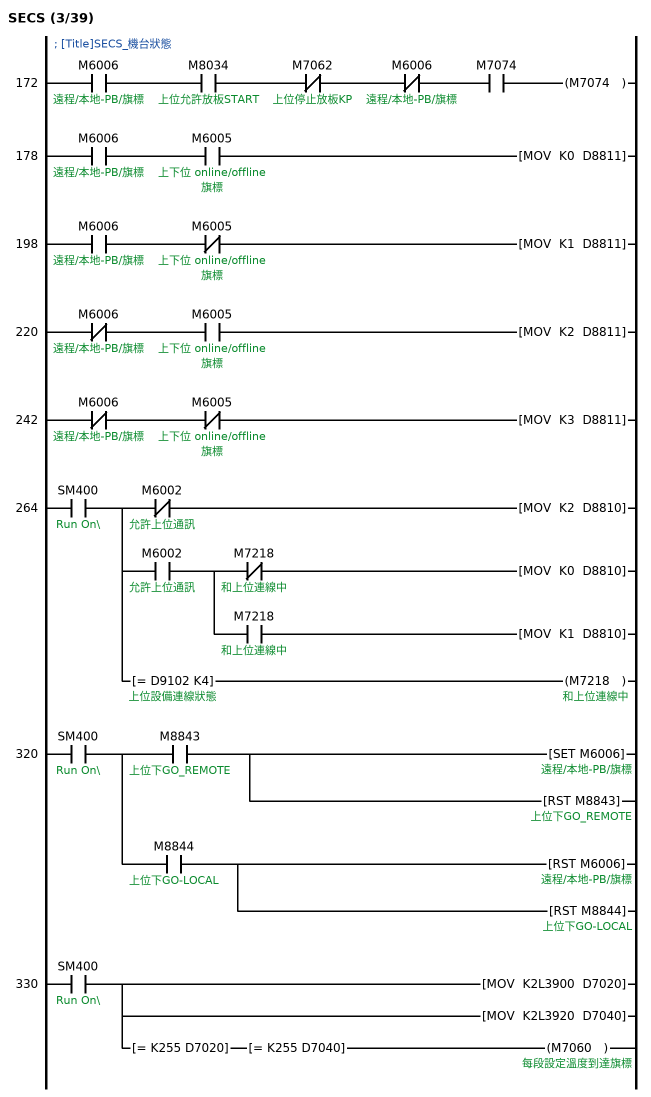
; [Title]SECS_機台狀態
172   LD      M6006  ; 遠程/本地-PB/旗標
      AND     M8034  ; 上位允許放板START
      ANI     M7062  ; 上位停止放板KP
      ANI     M6006  ; 遠程/本地-PB/旗標
      AND     M7074
      OUT     M7074
178   LD      M6006  ; 遠程/本地-PB/旗標
      AND     M6005  ; 上下位 online/offline 旗標
      MOV     K0 D8811
        [note] D8811=K0(遠程控制+SEC在線中)
198   LD      M6006  ; 遠程/本地-PB/旗標
      ANI     M6005  ; 上下位 online/offline 旗標
      MOV     K1 D8811
        [note] D8811= k1(遠程控制中+SEC離線中)
220   LDI     M6006  ; 遠程/本地-PB/旗標
      AND     M6005  ; 上下位 online/offline 旗標
      MOV     K2 D8811
        [note] D881=k2(遠程控制離線+SEC在線中)
242   LDI     M6006  ; 遠程/本地-PB/旗標
      ANI     M6005  ; 上下位 online/offline 旗標
      MOV     K3 D8811
        [note] D881=k3(遠程控制離線+SEC離線中)
264   LD      SM400  ; Run On\
      MPS
      ANI     M6002  ; 允許上位通訊
      MOV     K2 D8810
        [note] K2= SEC通訊未連線
      MRD
      AND     M6002  ; 允許上位通訊
      MPS
      ANI     M7218  ; 和上位連線中
      MOV     K0 D8810
        [note] K0=SEC連線---上位未連線
      MPP
      AND     M7218  ; 和上位連線中
      MOV     K1 D8810
        [note] K1=SEC和上位連線中
      MPP
      AND=    D9102 K4  ; 上位設備連線狀態
      OUT     M7218  ; 和上位連線中
320   LD      SM400  ; Run On\
      MPS
      AND     M8843  ; 上位下GO_REMOTE
      SET     M6006  ; 遠程/本地-PB/旗標
      RST     M8843  ; 上位下GO_REMOTE
      MPP
      AND     M8844  ; 上位下GO-LOCAL
      RST     M6006  ; 遠程/本地-PB/旗標
      RST     M8844  ; 上位下GO-LOCAL
330   LD      SM400  ; Run On\
      MOV     K2L3900 D7020  ; 溫度到達H01
      MOV     K2L3920 D7040  ; 溫度到達IRA01
      AND=    K255 D7020
      AND=    K255 D7040
      OUT     M7060  ; 每段設定溫度到達旗標
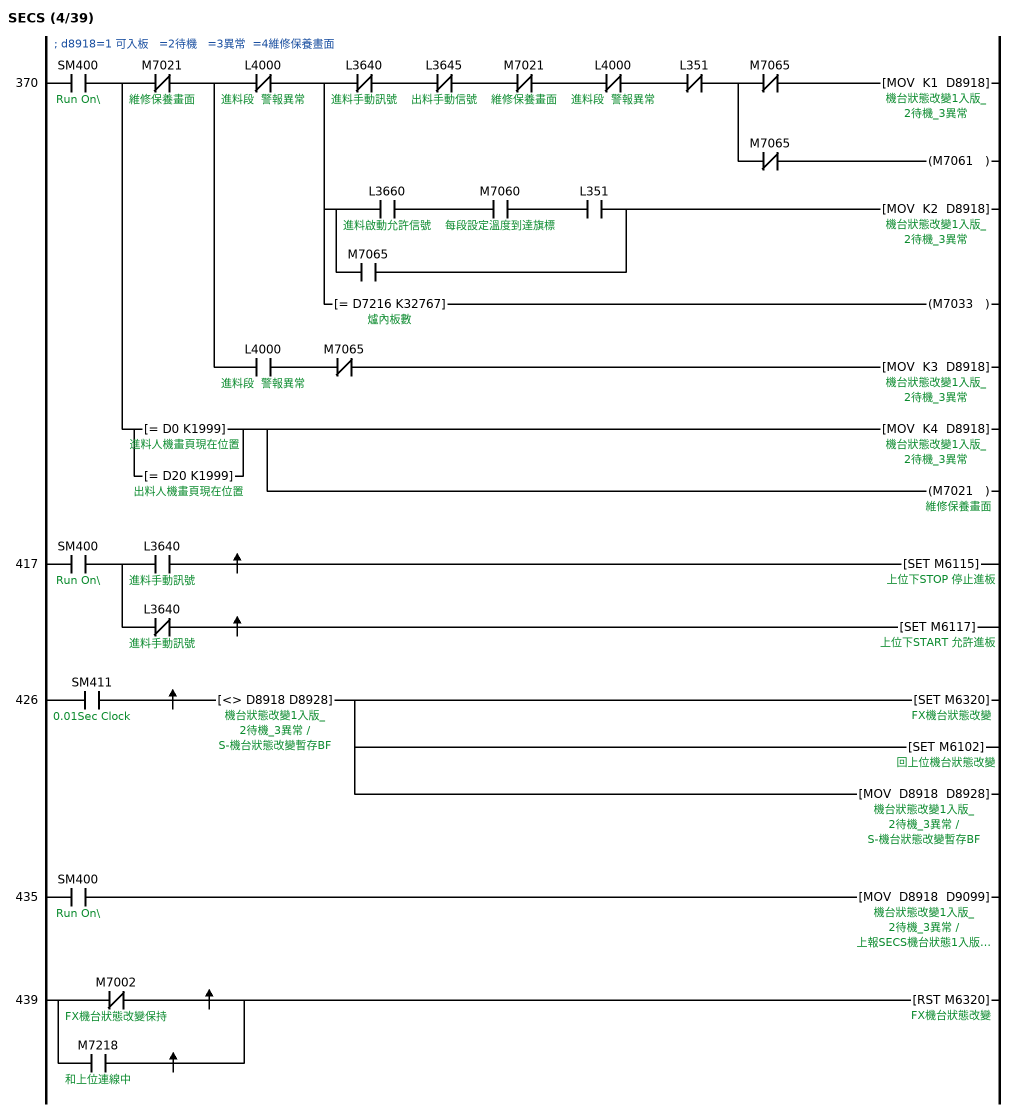
; d8918=1 可入板   =2待機   =3異常  =4維修保養畫面
370   LD      SM400  ; Run On\
      MPS
      ANI     M7021  ; 維修保養畫面
      MPS
      ANI     L4000  ; 進料段  警報異常
      MPS
      ANI     L3640  ; 進料手動訊號
      ANI     L3645  ; 出料手動信號
      ANI     M7021  ; 維修保養畫面
      ANI     L4000  ; 進料段  警報異常
      ANI     L351
      MPS
      ANI     M7065
      MOV     K1 D8918  ; 機台狀態改變1入版_2待機_3異常
      MPP
      ANI     M7065
      OUT     M7061
      MRD
      LD      L3660  ; 進料啟動允許信號
      AND     M7060  ; 每段設定溫度到達旗標
      AND     L351
      OR      M7065
      ANB
      MOV     K2 D8918
      MPP
      AND=    D7216 K32767  ; 爐內板數
      OUT     M7033
      MPP
      AND     L4000  ; 進料段  警報異常
      ANI     M7065
      MOV     K3 D8918
      MPP
      LD=     D0 K1999  ; 進料人機畫頁現在位置
      OR=     D20 K1999  ; 出料人機畫頁現在位置
      ANB
      MOV     K4 D8918
      OUT     M7021  ; 維修保養畫面
417   LD      SM400  ; Run On\
      MPS
      AND     L3640  ; 進料手動訊號
      MEP
      SET     M6115  ; 上位下STOP 停止進板
      MPP
      ANI     L3640  ; 進料手動訊號
      MEP
      SET     M6117  ; 上位下START 允許進板
426   LD      SM411  ; 0.01Sec Clock
      MEP
      AND<>   D8918 D8928  ; 機台狀態改變1入版_2待機_3異常 / S-機台狀態改變暫存BF
      SET     M6320  ; FX機台狀態改變
      SET     M6102  ; 回上位機台狀態改變
      MOV     D8918 D8928
435   LD      SM400  ; Run On\
      MOV     D8918 D9099  ; 上報SECS機台狀態1入版_2待機_3異
439   LDI     M7002  ; FX機台狀態改變保持
      MEP
      LD      M7218  ; 和上位連線中
      MEP
      ORB
      RST     M6320  ; FX機台狀態改變
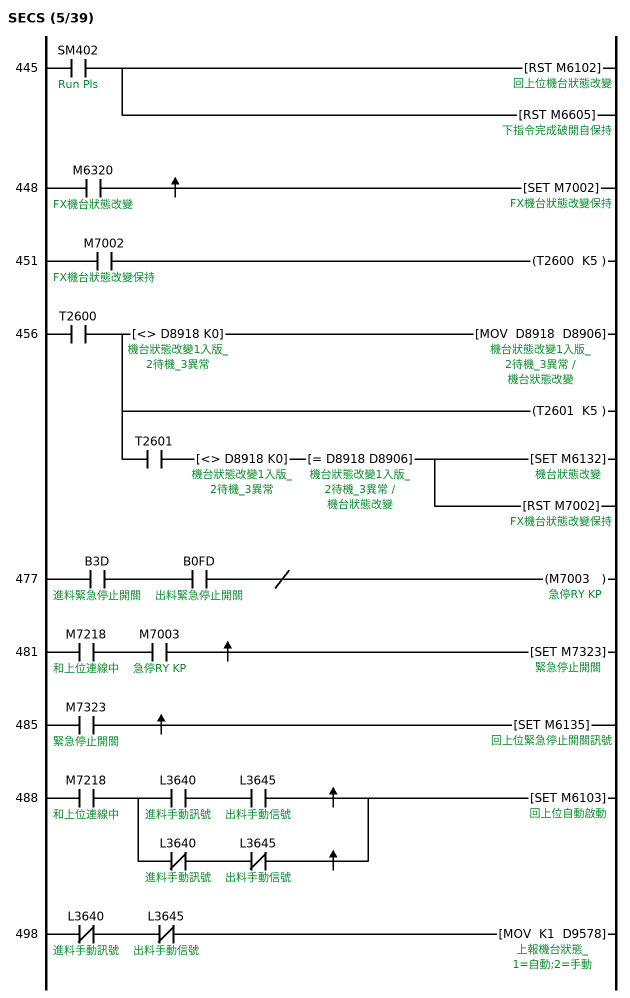
445   LD      SM402  ; Run Pls
      RST     M6102  ; 回上位機台狀態改變
      RST     M6605  ; 下指令完成破開自保持
448   LD      M6320  ; FX機台狀態改變
      MEP
      SET     M7002  ; FX機台狀態改變保持
451   LD      M7002  ; FX機台狀態改變保持
      OUT     T2600 K5
456   LD      T2600
      MPS
      AND<>   D8918 K0  ; 機台狀態改變1入版_2待機_3異常
      MOV     D8918 D8906  ; 機台狀態改變
      MPP
      OUT     T2601 K5
      AND     T2601
      AND<>   D8918 K0  ; 機台狀態改變1入版_2待機_3異常
      AND=    D8918 D8906  ; 機台狀態改變1入版_2待機_3異常 / 機台狀態改變
      SET     M6132  ; 機台狀態改變
      RST     M7002  ; FX機台狀態改變保持
477   LD      B3D  ; 進料緊急停止開關
      AND     B0FD  ; 出料緊急停止開關
      INV
      OUT     M7003  ; 急停RY KP
481   LD      M7218  ; 和上位連線中
      AND     M7003  ; 急停RY KP
      MEP
      SET     M7323  ; 緊急停止開關
485   LD      M7323  ; 緊急停止開關
      MEP
      SET     M6135  ; 回上位緊急停止開關訊號
488   LD      M7218  ; 和上位連線中
      LD      L3640  ; 進料手動訊號
      AND     L3645  ; 出料手動信號
      MEP
      LDI     L3640  ; 進料手動訊號
      ANI     L3645  ; 出料手動信號
      MEP
      ORB
      ANB
      SET     M6103  ; 回上位自動啟動
498   LDI     L3640  ; 進料手動訊號
      ANI     L3645  ; 出料手動信號
      MOV     K1 D9578  ; 上報機台狀態_1=自動;2=手動
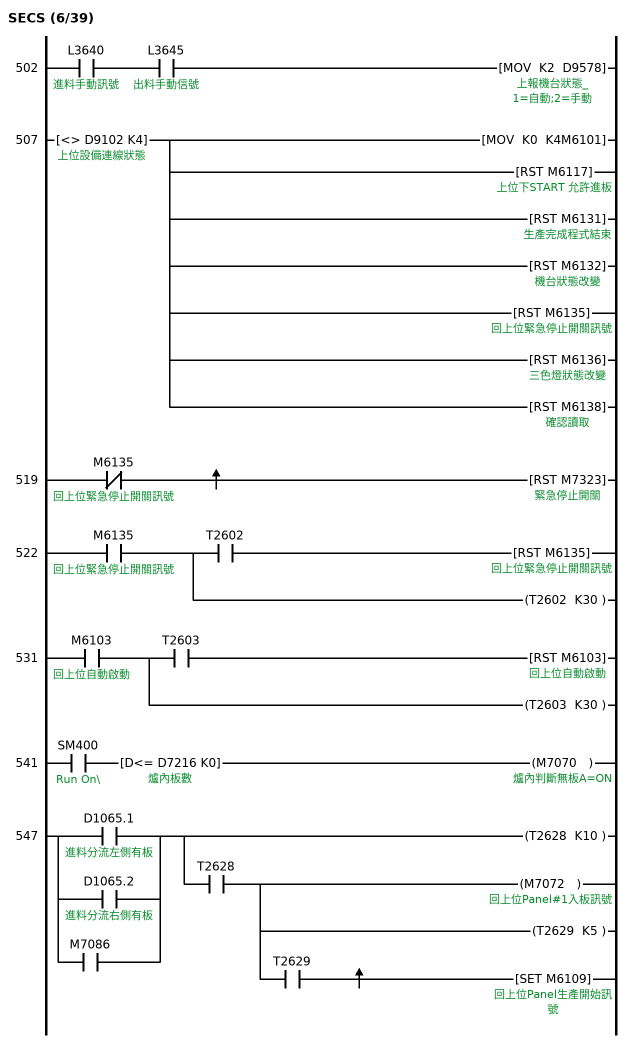
502   LD      L3640  ; 進料手動訊號
      AND     L3645  ; 出料手動信號
      MOV     K2 D9578
507   LD<>    D9102 K4  ; 上位設備連線狀態
      MOV     K0 K4M6101
      RST     M6117  ; 上位下START 允許進板
      RST     M6131  ; 生產完成程式結束
      RST     M6132  ; 機台狀態改變
      RST     M6135  ; 回上位緊急停止開關訊號
      RST     M6136  ; 三色燈狀態改變
      RST     M6138  ; 確認讀取
519   LDI     M6135  ; 回上位緊急停止開關訊號
      MEP
      RST     M7323  ; 緊急停止開關
522   LD      M6135  ; 回上位緊急停止開關訊號
      MPS
      AND     T2602
      RST     M6135  ; 回上位緊急停止開關訊號
      MPP
      OUT     T2602 K30
531   LD      M6103  ; 回上位自動啟動
      MPS
      AND     T2603
      RST     M6103  ; 回上位自動啟動
      MPP
      OUT     T2603 K30
541   LD      SM400  ; Run On\
      ANDD<=  D7216 K0  ; 爐內板數
      OUT     M7070  ; 爐內判斷無板A=ON
547   LD      D1065.1  ; 進料分流左側有板
      OR      D1065.2  ; 進料分流右側有板
      OR      M7086
      OUT     T2628 K10
      AND     T2628
      OUT     M7072  ; 回上位Panel#1入板訊號
      OUT     T2629 K5
      AND     T2629
      MEP
      SET     M6109  ; 回上位Panel生產開始訊號
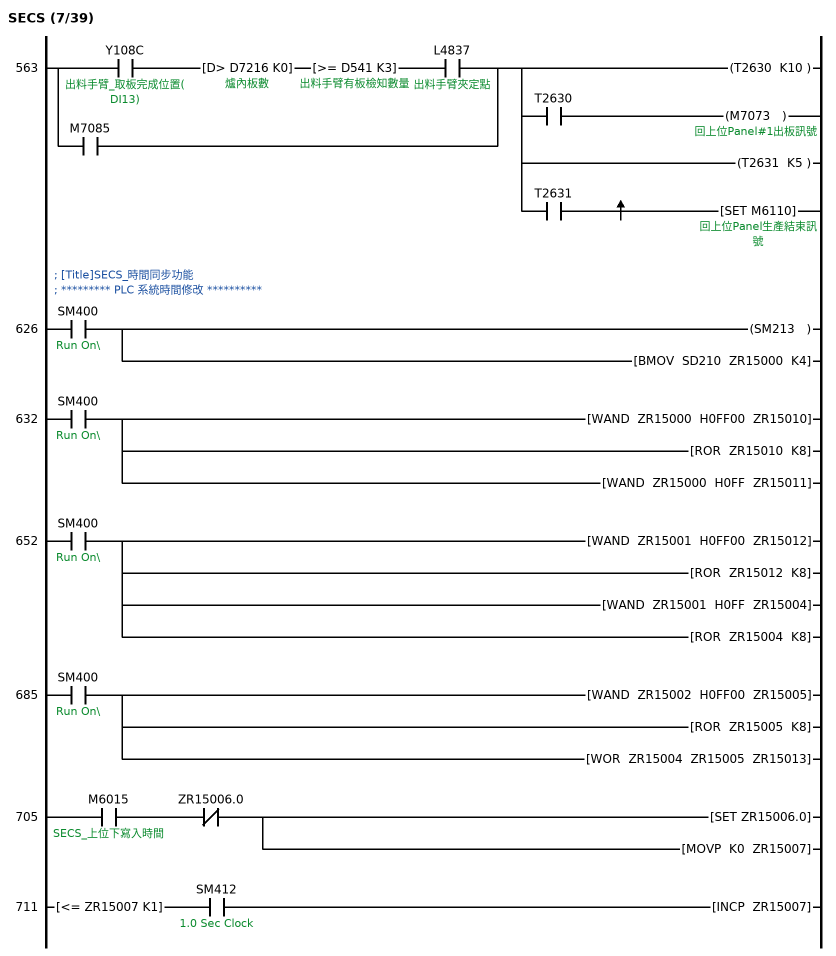
563   LD      Y108C  ; 出料手臂_取板完成位置(DI13)
      ANDD>   D7216 K0  ; 爐內板數
      AND>=   D541 K3  ; 出料手臂有板檢知數量
      AND     L4837  ; 出料手臂夾定點
      OR      M7085
      OUT     T2630 K10
      MPS
      AND     T2630
      OUT     M7073  ; 回上位Panel#1出板訊號
      MPP
      OUT     T2631 K5
      AND     T2631
      MEP
      SET     M6110  ; 回上位Panel生產結束訊號
; [Title]SECS_時間同步功能
; ********* PLC 系統時間修改 **********
626   LD      SM400  ; Run On\
      OUT     SM213
      BMOV    SD210 ZR15000 K4
632   LD      SM400  ; Run On\
      WAND    ZR15000 H0FF00 ZR15010
      ROR     ZR15010 K8
        [note] 高低位資料互換
      WAND    ZR15000 H0FF ZR15011
652   LD      SM400  ; Run On\
      WAND    ZR15001 H0FF00 ZR15012
      ROR     ZR15012 K8
        [note] 高低位資料互換
      WAND    ZR15001 H0FF ZR15004
      ROR     ZR15004 K8
        [note] 高低位資料互換
685   LD      SM400  ; Run On\
      WAND    ZR15002 H0FF00 ZR15005
      ROR     ZR15005 K8
        [note] 高低位資料互換
      WOR     ZR15004 ZR15005 ZR15013
705   LD      M6015  ; SECS_上位下寫入時間
      ANI     ZR15006.0
      SET     ZR15006.0
      MOVP    K0 ZR15007
711   LD<=    ZR15007 K1
      AND     SM412  ; 1.0 Sec Clock
      INCP    ZR15007
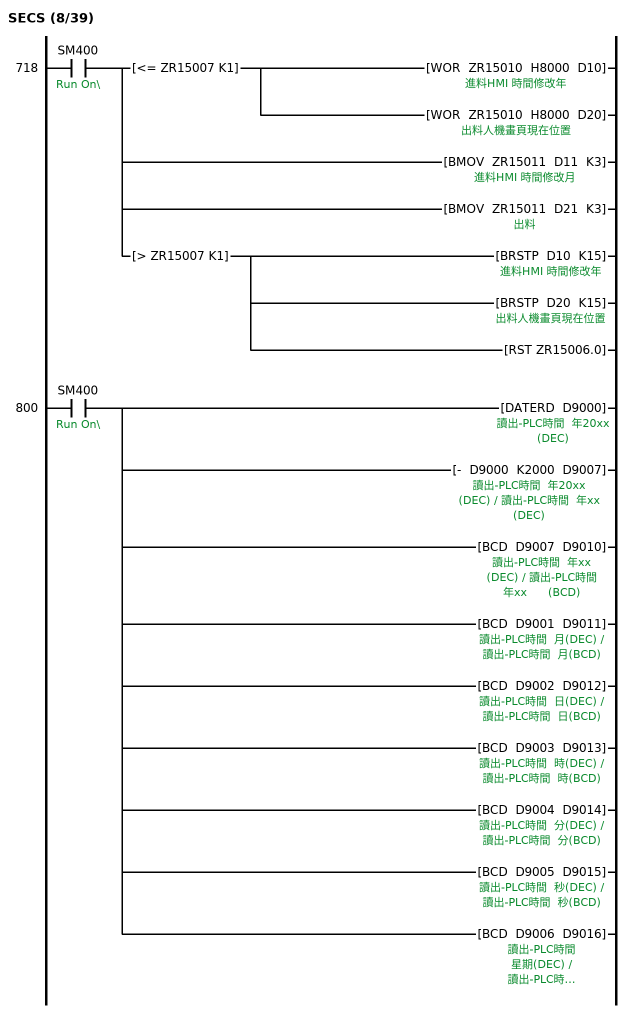
718   LD      SM400  ; Run On\
      MPS
      AND<=   ZR15007 K1
      WOR     ZR15010 H8000 D10  ; 進料HMI 時間修改年
        [note] HMI 時間修改命令H8000
      WOR     ZR15010 H8000 D20
        [note] HMI 時間修改命令H8000
      MPP
      BMOV    ZR15011 D11 K3  ; 進料HMI 時間修改月
      BMOV    ZR15011 D21 K3  ; 出料
      AND>    ZR15007 K1
      BRSTP   D10 K15
        [note] HMI 時間修改命令解除
      BRSTP   D20 K15
        [note] HMI 時間修改命令解除
      RST     ZR15006.0
800   LD      SM400  ; Run On\
      DATERD  D9000  ; 讀出-PLC時間  年20xx    (DEC)
      -       D9000 K2000 D9007  ; 讀出-PLC時間  年xx      (DEC)
      BCD     D9007 D9010  ; 讀出-PLC時間  年xx      (BCD)
      BCD     D9001 D9011  ; 讀出-PLC時間  月(DEC) / 讀出-PLC時間  月(BCD)
      BCD     D9002 D9012  ; 讀出-PLC時間  日(DEC) / 讀出-PLC時間  日(BCD)
      BCD     D9003 D9013  ; 讀出-PLC時間  時(DEC) / 讀出-PLC時間  時(BCD)
      BCD     D9004 D9014  ; 讀出-PLC時間  分(DEC) / 讀出-PLC時間  分(BCD)
      BCD     D9005 D9015  ; 讀出-PLC時間  秒(DEC) / 讀出-PLC時間  秒(BCD)
      BCD     D9006 D9016  ; 讀出-PLC時間  星期(DEC) / 讀出-PLC時間  星期(BCD)
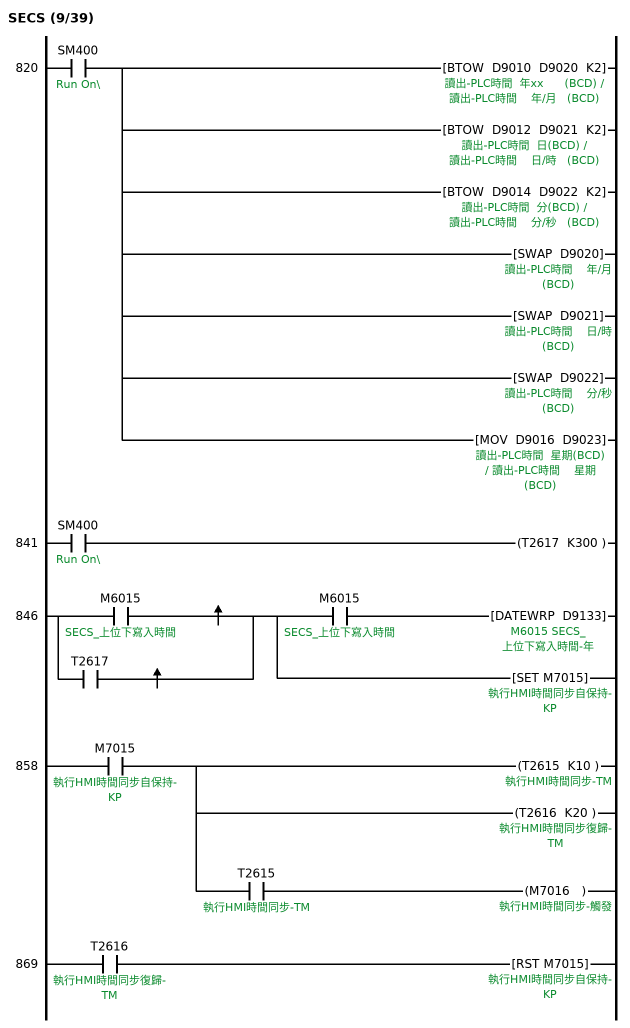
820   LD      SM400  ; Run On\
      BTOW    D9010 D9020 K2  ; 讀出-PLC時間    年/月   (BCD)
      BTOW    D9012 D9021 K2  ; 讀出-PLC時間    日/時   (BCD)
      BTOW    D9014 D9022 K2  ; 讀出-PLC時間    分/秒   (BCD)
      SWAP    D9020
      SWAP    D9021
      SWAP    D9022
      MOV     D9016 D9023  ; 讀出-PLC時間    星期    (BCD)
841   LD      SM400  ; Run On\
      OUT     T2617 K300
846   LD      M6015  ; SECS_上位下寫入時間
      MEP
      LD      T2617
      MEP
      ORB
      MPS
      AND     M6015  ; SECS_上位下寫入時間
      DATEWRP D9133  ; M6015 SECS_上位下寫入時間-年
      MPP
      SET     M7015  ; 執行HMI時間同步自保持-KP
858   LD      M7015  ; 執行HMI時間同步自保持-KP
      OUT     T2615 K10  ; 執行HMI時間同步-TM
      OUT     T2616 K20  ; 執行HMI時間同步復歸-TM
      AND     T2615  ; 執行HMI時間同步-TM
      OUT     M7016  ; 執行HMI時間同步-觸發
869   LD      T2616  ; 執行HMI時間同步復歸-TM
      RST     M7015  ; 執行HMI時間同步自保持-KP
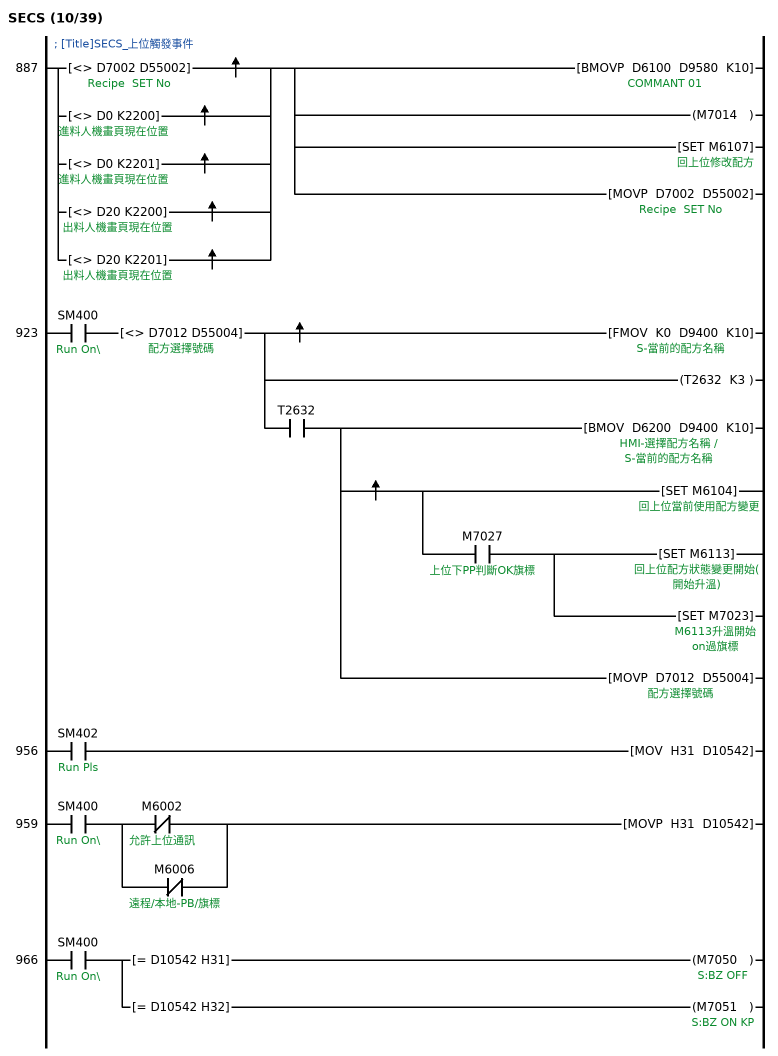
; [Title]SECS_上位觸發事件
887   LD<>    D7002 D55002  ; Recipe  SET No
      MEP
      LD<>    D0 K2200  ; 進料人機畫頁現在位置
      MEP
      ORB
      LD<>    D0 K2201  ; 進料人機畫頁現在位置
      MEP
      ORB
      LD<>    D20 K2200  ; 出料人機畫頁現在位置
      MEP
      ORB
      LD<>    D20 K2201  ; 出料人機畫頁現在位置
      MEP
      ORB
      BMOVP   D6100 D9580 K10  ; COMMANT 01
      OUT     M7014
      SET     M6107  ; 回上位修改配方
      MOVP    D7002 D55002
923   LD      SM400  ; Run On\
      AND<>   D7012 D55004  ; 配方選擇號碼
      MPS
      MEP
      FMOV    K0 D9400 K10  ; S-當前的配方名稱
      MPP
      OUT     T2632 K3
      AND     T2632
      BMOV    D6200 D9400 K10  ; HMI-選擇配方名稱
      MPS
      MEP
      SET     M6104  ; 回上位當前使用配方變更
      AND     M7027  ; 上位下PP判斷OK旗標
      SET     M6113  ; 回上位配方狀態變更開始(開始升溫)
      SET     M7023  ; M6113升溫開始 on過旗標
      MPP
      MOVP    D7012 D55004
956   LD      SM402  ; Run Pls
      MOV     H31 D10542
959   LD      SM400  ; Run On\
      LDI     M6002  ; 允許上位通訊
      ORI     M6006  ; 遠程/本地-PB/旗標
      ANB
      MOVP    H31 D10542
966   LD      SM400  ; Run On\
      MPS
      AND=    D10542 H31
      OUT     M7050  ; S:BZ OFF
      MPP
      AND=    D10542 H32
      OUT     M7051  ; S:BZ ON KP
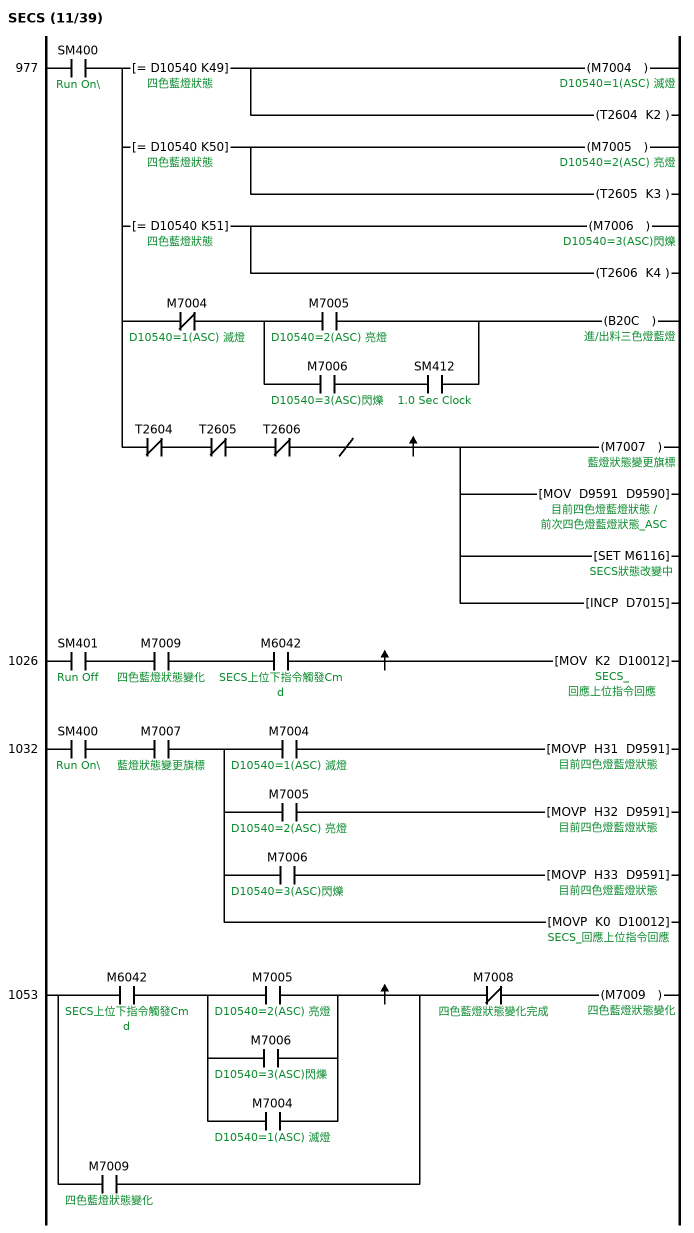
977   LD      SM400  ; Run On\
      MPS
      AND=    D10540 K49  ; 四色藍燈狀態
      OUT     M7004  ; D10540=1(ASC) 滅燈
      OUT     T2604 K2
      MRD
      AND=    D10540 K50  ; 四色藍燈狀態
      OUT     M7005  ; D10540=2(ASC) 亮燈
      OUT     T2605 K3
      MRD
      AND=    D10540 K51  ; 四色藍燈狀態
      OUT     M7006  ; D10540=3(ASC)閃爍
      OUT     T2606 K4
      MRD
      ANI     M7004  ; D10540=1(ASC) 滅燈
      LD      M7005  ; D10540=2(ASC) 亮燈
      LD      M7006  ; D10540=3(ASC)閃爍
      AND     SM412  ; 1.0 Sec Clock
      ORB
      ANB
      OUT     B20C  ; 進/出料三色燈藍燈
      MPP
      ANI     T2604
      ANI     T2605
      ANI     T2606
      INV
      MEP
      OUT     M7007  ; 藍燈狀態變更旗標
      MOV     D9591 D9590  ; 目前四色燈藍燈狀態 / 前次四色燈藍燈狀態_ASC
      SET     M6116  ; SECS狀態改變中
      INCP    D7015
1026  LD      SM401  ; Run Off
      AND     M7009  ; 四色藍燈狀態變化
      AND     M6042  ; SECS上位下指令觸發Cmd
      MEP
      MOV     K2 D10012  ; SECS_回應上位指令回應
1032  LD      SM400  ; Run On\
      AND     M7007  ; 藍燈狀態變更旗標
      MPS
      AND     M7004  ; D10540=1(ASC) 滅燈
      MOVP    H31 D9591
      MRD
      AND     M7005  ; D10540=2(ASC) 亮燈
      MOVP    H32 D9591
      MRD
      AND     M7006  ; D10540=3(ASC)閃爍
      MOVP    H33 D9591
      MPP
      MOVP    K0 D10012
1053  LD      M6042  ; SECS上位下指令觸發Cmd
      LD      M7005  ; D10540=2(ASC) 亮燈
      OR      M7006  ; D10540=3(ASC)閃爍
      OR      M7004  ; D10540=1(ASC) 滅燈
      ANB
      MEP
      OR      M7009  ; 四色藍燈狀態變化
      ANI     M7008  ; 四色藍燈狀態變化完成
      OUT     M7009  ; 四色藍燈狀態變化
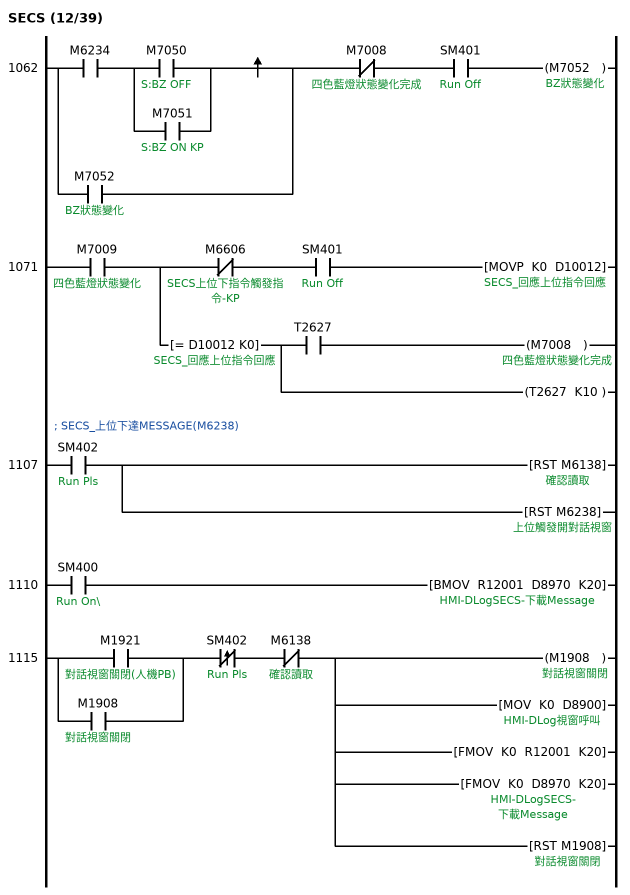
1062  LD      M6234
      LD      M7050  ; S:BZ OFF
      OR      M7051  ; S:BZ ON KP
      ANB
      MEP
      OR      M7052  ; BZ狀態變化
      ANI     M7008  ; 四色藍燈狀態變化完成
      AND     SM401  ; Run Off
      OUT     M7052  ; BZ狀態變化
1071  LD      M7009  ; 四色藍燈狀態變化
      MPS
      ANI     M6606  ; SECS上位下指令觸發指令-KP
      AND     SM401  ; Run Off
      MOVP    K0 D10012
      MPP
      AND=    D10012 K0  ; SECS_回應上位指令回應
      MPS
      AND     T2627
      OUT     M7008  ; 四色藍燈狀態變化完成
      MPP
      OUT     T2627 K10
; SECS_上位下達MESSAGE(M6238)
1107  LD      SM402  ; Run Pls
      RST     M6138  ; 確認讀取
      RST     M6238  ; 上位觸發開對話視窗
1110  LD      SM400  ; Run On\
      BMOV    R12001 D8970 K20  ; HMI-DLogSECS-下載Message
1115  LD      M1921  ; 對話視窗關閉(人機PB)
      OR      M1908  ; 對話視窗關閉
      ANDPI   SM402  ; Run Pls
      ANI     M6138  ; 確認讀取
      OUT     M1908  ; 對話視窗關閉
      MOV     K0 D8900  ; HMI-DLog視窗呼叫
      FMOV    K0 R12001 K20
      FMOV    K0 D8970 K20
      RST     M1908  ; 對話視窗關閉
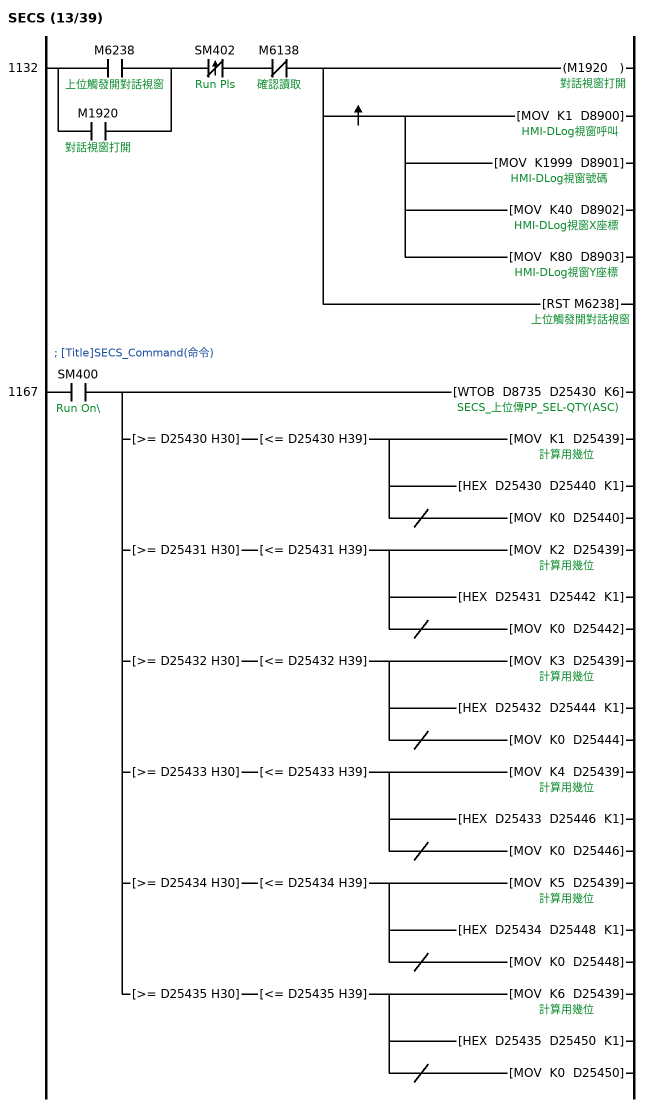
1132  LD      M6238  ; 上位觸發開對話視窗
      OR      M1920  ; 對話視窗打開
      ANDPI   SM402  ; Run Pls
      ANI     M6138  ; 確認讀取
      OUT     M1920  ; 對話視窗打開
      MPS
      MEP
      MOV     K1 D8900
      MOV     K1999 D8901  ; HMI-DLog視窗號碼
      MOV     K40 D8902  ; HMI-DLog視窗X座標
      MOV     K80 D8903  ; HMI-DLog視窗Y座標
      MPP
      RST     M6238  ; 上位觸發開對話視窗
; [Title]SECS_Command(命令)
1167  LD      SM400  ; Run On\
      WTOB    D8735 D25430 K6  ; SECS_上位傳PP_SEL-QTY(ASC)
      MPS
      AND>=   D25430 H30
      AND<=   D25430 H39
      MOV     K1 D25439  ; 計算用幾位
      HEX     D25430 D25440 K1
      INV
      MOV     K0 D25440
      MRD
      AND>=   D25431 H30
      AND<=   D25431 H39
      MOV     K2 D25439
      HEX     D25431 D25442 K1
      INV
      MOV     K0 D25442
      MRD
      AND>=   D25432 H30
      AND<=   D25432 H39
      MOV     K3 D25439
      HEX     D25432 D25444 K1
      INV
      MOV     K0 D25444
      MRD
      AND>=   D25433 H30
      AND<=   D25433 H39
      MOV     K4 D25439
      HEX     D25433 D25446 K1
      INV
      MOV     K0 D25446
      MRD
      AND>=   D25434 H30
      AND<=   D25434 H39
      MOV     K5 D25439
      HEX     D25434 D25448 K1
      INV
      MOV     K0 D25448
      MPP
      AND>=   D25435 H30
      AND<=   D25435 H39
      MOV     K6 D25439
      HEX     D25435 D25450 K1
      INV
      MOV     K0 D25450
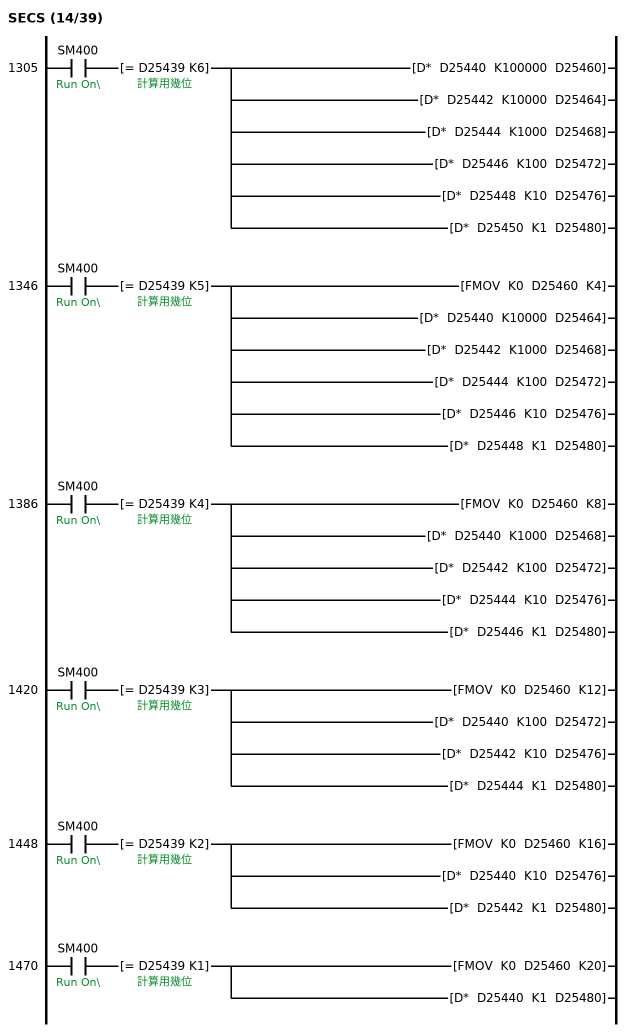
1305  LD      SM400  ; Run On\
      AND=    D25439 K6  ; 計算用幾位
      D*      D25440 K100000 D25460
      D*      D25442 K10000 D25464
      D*      D25444 K1000 D25468
      D*      D25446 K100 D25472
      D*      D25448 K10 D25476
      D*      D25450 K1 D25480
1346  LD      SM400  ; Run On\
      AND=    D25439 K5  ; 計算用幾位
      FMOV    K0 D25460 K4
      D*      D25440 K10000 D25464
      D*      D25442 K1000 D25468
      D*      D25444 K100 D25472
      D*      D25446 K10 D25476
      D*      D25448 K1 D25480
1386  LD      SM400  ; Run On\
      AND=    D25439 K4  ; 計算用幾位
      FMOV    K0 D25460 K8
      D*      D25440 K1000 D25468
      D*      D25442 K100 D25472
      D*      D25444 K10 D25476
      D*      D25446 K1 D25480
1420  LD      SM400  ; Run On\
      AND=    D25439 K3  ; 計算用幾位
      FMOV    K0 D25460 K12
      D*      D25440 K100 D25472
      D*      D25442 K10 D25476
      D*      D25444 K1 D25480
1448  LD      SM400  ; Run On\
      AND=    D25439 K2  ; 計算用幾位
      FMOV    K0 D25460 K16
      D*      D25440 K10 D25476
      D*      D25442 K1 D25480
1470  LD      SM400  ; Run On\
      AND=    D25439 K1  ; 計算用幾位
      FMOV    K0 D25460 K20
      D*      D25440 K1 D25480
